  MoveL 6051 to (232.86, 162.69, 88.06) mm, rotated rx 180 ry 0 rz 180 deg; joints [-65.874, 60.657, -79.327, 67.008, 97.518, 17.138]
  Call Extruder(269.01860)
  MoveL 6052 to (232.62, 162.8, 88.06) mm, rotated rx 180 ry 0 rz 180 deg; joints [-65.961, 60.657, -79.327, 67.092, 97.493, 17.15]
  MoveL 6053 to (232.62, 162.8, 88.06) mm, rotated rx 180 ry 0 rz 180 deg; joints [-65.961, 60.657, -79.327, 67.092, 97.493, 17.15]
  Call Extruder(269.17597)
  MoveL 6054 to (232.37, 162.91, 88.06) mm, rotated rx -180 ry 0 rz 180 deg; joints [-66.048, 60.657, -79.327, 67.176, 97.467, 17.161]
  MoveL 6055 to (232.37, 162.91, 88.06) mm, rotated rx -180 ry 0 rz 180 deg; joints [-66.048, 60.657, -79.327, 67.176, 97.467, 17.161]
  Call Extruder(269.35871)
  MoveL 6056 to (232.07, 163.02, 88.06) mm, rotated rx -180 ry 0 rz -180 deg; joints [-66.149, 60.656, -79.328, 67.274, 97.438, 17.175]
  MoveL 6057 to (232.07, 163.02, 88.06) mm, rotated rx -180 ry 0 rz -180 deg; joints [-66.149, 60.656, -79.328, 67.274, 97.438, 17.175]
  Call Extruder(269.54070)
  MoveL 6058 to (231.78, 163.15, 88.06) mm, rotated rx 180 ry 0 rz 180 deg; joints [-66.251, 60.655, -79.328, 67.372, 97.408, 17.188]
  MoveL 6059 to (231.78, 163.15, 88.06) mm, rotated rx 180 ry 0 rz 180 deg; joints [-66.251, 60.655, -79.328, 67.372, 97.408, 17.188]
  Call Extruder(269.68804)
  MoveL 6060 to (231.54, 163.24, 88.06) mm, rotated rx -180 ry 0 rz -180 deg; joints [-66.333, 60.654, -79.328, 67.452, 97.384, 17.2]
  MoveL 6061 to (231.54, 163.24, 88.06) mm, rotated rx -180 ry 0 rz -180 deg; joints [-66.333, 60.654, -79.328, 67.452, 97.384, 17.2]
  Call Extruder(269.80126)
  MoveL 6062 to (231.35, 163.3, 88.06) mm, rotated rx 180 ry 0 rz -180 deg; joints [-66.397, 60.653, -79.329, 67.513, 97.367, 17.21]
  MoveL 6063 to (231.35, 163.3, 88.06) mm, rotated rx 180 ry 0 rz -180 deg; joints [-66.397, 60.653, -79.329, 67.513, 97.367, 17.21]
  Call Extruder(269.91404)
  MoveL 6064 to (231.17, 163.36, 88.06) mm, rotated rx 180 ry 0 rz -180 deg; joints [-66.46, 60.651, -79.33, 67.574, 97.349, 17.22]
  MoveL 6065 to (231.17, 163.36, 88.06) mm, rotated rx 180 ry 0 rz -180 deg; joints [-66.46, 60.651, -79.33, 67.574, 97.349, 17.22]
  Call Extruder(270.02637)
  MoveL 6066 to (230.98, 163.42, 88.06) mm, rotated rx -180 ry 0 rz 180 deg; joints [-66.524, 60.65, -79.331, 67.636, 97.331, 17.23]
  MoveL 6067 to (230.98, 163.42, 88.06) mm, rotated rx -180 ry 0 rz 180 deg; joints [-66.524, 60.65, -79.331, 67.636, 97.331, 17.23]
  Call Extruder(270.13826)
  MoveL 6068 to (230.79, 163.48, 88.06) mm, rotated rx -180 ry 0 rz 180 deg; joints [-66.587, 60.648, -79.331, 67.697, 97.313, 17.24]
  MoveL 6069 to (230.79, 163.48, 88.06) mm, rotated rx -180 ry 0 rz 180 deg; joints [-66.587, 60.648, -79.331, 67.697, 97.313, 17.24]
  Call Extruder(270.25966)
  MoveL 6070 to (230.58, 163.55, 88.06) mm, rotated rx -180 ry 0 rz -180 deg; joints [-66.656, 60.646, -79.332, 67.764, 97.293, 17.251]
  MoveL 6071 to (230.58, 163.55, 88.06) mm, rotated rx -180 ry 0 rz -180 deg; joints [-66.656, 60.646, -79.332, 67.764, 97.293, 17.251]
  Call Extruder(270.39048)
  MoveL 6072 to (230.36, 163.62, 88.06) mm, rotated rx -180 ry 0 rz 180 deg; joints [-66.731, 60.644, -79.333, 67.836, 97.272, 17.263]
  MoveL 6073 to (230.36, 163.62, 88.06) mm, rotated rx -180 ry 0 rz 180 deg; joints [-66.731, 60.644, -79.333, 67.836, 97.272, 17.263]
  Call Extruder(270.52072)
  MoveL 6074 to (230.14, 163.68, 88.06) mm, rotated rx 180 ry 0 rz 180 deg; joints [-66.805, 60.642, -79.334, 67.908, 97.251, 17.275]
  MoveL 6075 to (230.14, 163.68, 88.06) mm, rotated rx 180 ry 0 rz 180 deg; joints [-66.805, 60.642, -79.334, 67.908, 97.251, 17.275]
  Call Extruder(270.65041)
  MoveL 6076 to (229.91, 163.75, 88.06) mm, rotated rx 180 ry 0 rz -180 deg; joints [-66.88, 60.64, -79.335, 67.981, 97.23, 17.287]
  MoveL 6077 to (229.91, 163.75, 88.06) mm, rotated rx 180 ry 0 rz -180 deg; joints [-66.88, 60.64, -79.335, 67.981, 97.23, 17.287]
  Call Extruder(270.77952)
  MoveL 6078 to (229.69, 163.82, 88.06) mm, rotated rx -180 ry 0 rz 180 deg; joints [-66.955, 60.638, -79.336, 68.053, 97.209, 17.299]
  MoveL 6079 to (229.69, 163.82, 88.06) mm, rotated rx -180 ry 0 rz 180 deg; joints [-66.955, 60.638, -79.336, 68.053, 97.209, 17.299]
  Call Extruder(270.89460)
  MoveL 6080 to (229.48, 163.86, 88.06) mm, rotated rx 180 ry 0 rz 180 deg; joints [-67.021, 60.635, -79.338, 68.117, 97.191, 17.311]
  MoveL 6081 to (229.48, 163.86, 88.06) mm, rotated rx 180 ry 0 rz 180 deg; joints [-67.021, 60.635, -79.338, 68.117, 97.191, 17.311]
  Call Extruder(271.00922)
  MoveL 6082 to (229.28, 163.91, 88.06) mm, rotated rx -180 ry 0 rz 180 deg; joints [-67.087, 60.632, -79.339, 68.181, 97.173, 17.323]
  MoveL 6083 to (229.28, 163.91, 88.06) mm, rotated rx -180 ry 0 rz 180 deg; joints [-67.087, 60.632, -79.339, 68.181, 97.173, 17.323]
  Call Extruder(271.12339)
  MoveL 6084 to (229.08, 163.95, 88.06) mm, rotated rx 180 ry 0 rz -180 deg; joints [-67.153, 60.628, -79.341, 68.246, 97.155, 17.336]
  MoveL 6085 to (229.08, 163.95, 88.06) mm, rotated rx 180 ry 0 rz -180 deg; joints [-67.153, 60.628, -79.341, 68.246, 97.155, 17.336]
  Call Extruder(271.23711)
  MoveL 6086 to (228.87, 164, 88.06) mm, rotated rx 180 ry 0 rz -180 deg; joints [-67.22, 60.625, -79.342, 68.31, 97.137, 17.348]
  MoveL 6087 to (228.87, 164, 88.06) mm, rotated rx 180 ry 0 rz -180 deg; joints [-67.22, 60.625, -79.342, 68.31, 97.137, 17.348]
  Call Extruder(271.36253)
  MoveL 6088 to (228.64, 164.04, 88.06) mm, rotated rx -180 ry 0 rz -180 deg; joints [-67.293, 60.622, -79.344, 68.381, 97.118, 17.362]
  MoveL 6089 to (228.64, 164.04, 88.06) mm, rotated rx -180 ry 0 rz -180 deg; joints [-67.293, 60.622, -79.344, 68.381, 97.118, 17.362]
  Call Extruder(271.49950)
  MoveL 6090 to (228.4, 164.09, 88.06) mm, rotated rx -180 ry 0 rz -180 deg; joints [-67.373, 60.618, -79.346, 68.459, 97.096, 17.377]
  MoveL 6091 to (228.4, 164.09, 88.06) mm, rotated rx -180 ry 0 rz -180 deg; joints [-67.373, 60.618, -79.346, 68.459, 97.096, 17.377]
  Call Extruder(271.63587)
  MoveL 6092 to (228.15, 164.14, 88.06) mm, rotated rx -180 ry 0 rz 180 deg; joints [-67.453, 60.614, -79.348, 68.537, 97.074, 17.392]
  MoveL 6093 to (228.15, 164.14, 88.06) mm, rotated rx -180 ry 0 rz 180 deg; joints [-67.453, 60.614, -79.348, 68.537, 97.074, 17.392]
  Call Extruder(271.77163)
  MoveL 6094 to (227.9, 164.19, 88.06) mm, rotated rx -180 ry 0 rz -180 deg; joints [-67.534, 60.61, -79.35, 68.615, 97.052, 17.407]
  MoveL 6095 to (227.9, 164.19, 88.06) mm, rotated rx -180 ry 0 rz -180 deg; joints [-67.534, 60.61, -79.35, 68.615, 97.052, 17.407]
  Call Extruder(271.90678)
  MoveL 6096 to (227.65, 164.24, 88.06) mm, rotated rx -180 ry 0 rz 180 deg; joints [-67.614, 60.605, -79.352, 68.693, 97.03, 17.422]
  MoveL 6097 to (227.65, 164.24, 88.06) mm, rotated rx -180 ry 0 rz 180 deg; joints [-67.614, 60.605, -79.352, 68.693, 97.03, 17.422]
  Call Extruder(272.04131)
  MoveL 6098 to (227.4, 164.29, 88.06) mm, rotated rx -180 ry 0 rz 180 deg; joints [-67.695, 60.602, -79.354, 68.771, 97.008, 17.437]
  MoveL 6099 to (227.4, 164.29, 88.06) mm, rotated rx -180 ry 0 rz 180 deg; joints [-67.695, 60.602, -79.354, 68.771, 97.008, 17.437]
  Call Extruder(272.17524)
  MoveL 6100 to (227.15, 164.34, 88.06) mm, rotated rx 180 ry 0 rz -180 deg; joints [-67.775, 60.598, -79.355, 68.848, 96.986, 17.452]
  MoveL 6101 to (227.15, 164.34, 88.06) mm, rotated rx 180 ry 0 rz -180 deg; joints [-67.775, 60.598, -79.355, 68.848, 96.986, 17.452]
  Call Extruder(272.32310)
  MoveL 6102 to (226.87, 164.39, 88.06) mm, rotated rx 180 ry 0 rz 180 deg; joints [-67.864, 60.593, -79.358, 68.935, 96.962, 17.469]
  MoveL 6103 to (226.87, 164.39, 88.06) mm, rotated rx 180 ry 0 rz 180 deg; joints [-67.864, 60.593, -79.358, 68.935, 96.962, 17.469]
  Call Extruder(272.48484)
  MoveL 6104 to (226.57, 164.44, 88.06) mm, rotated rx -180 ry 0 rz -180 deg; joints [-67.961, 60.587, -79.36, 69.029, 96.936, 17.488]
  MoveL 6105 to (226.57, 164.44, 88.06) mm, rotated rx -180 ry 0 rz -180 deg; joints [-67.961, 60.587, -79.36, 69.029, 96.936, 17.488]
  Call Extruder(272.64586)
  MoveL 6106 to (226.26, 164.49, 88.06) mm, rotated rx -180 ry 0 rz -180 deg; joints [-68.059, 60.581, -79.363, 69.124, 96.91, 17.507]
  MoveL 6107 to (226.26, 164.49, 88.06) mm, rotated rx -180 ry 0 rz -180 deg; joints [-68.059, 60.581, -79.363, 69.124, 96.91, 17.507]
  Call Extruder(272.80614)
  MoveL 6108 to (225.96, 164.53, 88.06) mm, rotated rx -180 ry 0 rz 180 deg; joints [-68.156, 60.576, -79.366, 69.219, 96.883, 17.526]
  MoveL 6109 to (225.96, 164.53, 88.06) mm, rotated rx -180 ry 0 rz 180 deg; joints [-68.156, 60.576, -79.366, 69.219, 96.883, 17.526]
  Call Extruder(272.96570)
  MoveL 6110 to (225.65, 164.58, 88.06) mm, rotated rx -180 ry 0 rz 180 deg; joints [-68.254, 60.57, -79.368, 69.313, 96.857, 17.545]
  MoveL 6111 to (225.65, 164.58, 88.06) mm, rotated rx -180 ry 0 rz 180 deg; joints [-68.254, 60.57, -79.368, 69.313, 96.857, 17.545]
  Call Extruder(273.12452)
  MoveL 6112 to (225.34, 164.63, 88.06) mm, rotated rx 180 ry 0 rz 180 deg; joints [-68.351, 60.565, -79.371, 69.408, 96.83, 17.564]
  MoveL 6113 to (225.34, 164.63, 88.06) mm, rotated rx 180 ry 0 rz 180 deg; joints [-68.351, 60.565, -79.371, 69.408, 96.83, 17.564]
  Call Extruder(273.30319)
  MoveL 6114 to (225, 164.68, 88.06) mm, rotated rx 180 ry 0 rz 180 deg; joints [-68.461, 60.558, -79.374, 69.515, 96.801, 17.586]
  MoveL 6115 to (225, 164.68, 88.06) mm, rotated rx 180 ry 0 rz 180 deg; joints [-68.461, 60.558, -79.374, 69.515, 96.801, 17.586]
  Call Extruder(273.50164)
  MoveL 6116 to (224.61, 164.72, 88.06) mm, rotated rx -180 ry 0 rz 180 deg; joints [-68.583, 60.55, -79.378, 69.633, 96.768, 17.611]
  MoveL 6117 to (224.61, 164.72, 88.06) mm, rotated rx -180 ry 0 rz 180 deg; joints [-68.583, 60.55, -79.378, 69.633, 96.768, 17.611]
  Call Extruder(273.69921)
  MoveL 6118 to (224.22, 164.77, 88.06) mm, rotated rx -180 ry 0 rz 180 deg; joints [-68.706, 60.542, -79.382, 69.752, 96.735, 17.636]
  MoveL 6119 to (224.22, 164.77, 88.06) mm, rotated rx -180 ry 0 rz 180 deg; joints [-68.706, 60.542, -79.382, 69.752, 96.735, 17.636]
  Call Extruder(273.89592)
  MoveL 6120 to (223.84, 164.82, 88.06) mm, rotated rx 180 ry 0 rz 180 deg; joints [-68.828, 60.534, -79.386, 69.871, 96.702, 17.661]
  MoveL 6121 to (223.84, 164.82, 88.06) mm, rotated rx 180 ry 0 rz 180 deg; joints [-68.828, 60.534, -79.386, 69.871, 96.702, 17.661]
  Call Extruder(274.09176)
  MoveL 6122 to (223.45, 164.86, 88.06) mm, rotated rx -180 ry 0 rz 180 deg; joints [-68.951, 60.526, -79.389, 69.989, 96.669, 17.686]
  MoveL 6123 to (223.45, 164.86, 88.06) mm, rotated rx -180 ry 0 rz 180 deg; joints [-68.951, 60.526, -79.389, 69.989, 96.669, 17.686]
  Call Extruder(274.38712)
  MoveL 6124 to (222.86, 164.91, 88.06) mm, rotated rx -180 ry 0 rz 180 deg; joints [-69.135, 60.512, -79.396, 70.168, 96.62, 17.725]
  MoveL 6125 to (222.86, 164.91, 88.06) mm, rotated rx -180 ry 0 rz 180 deg; joints [-69.135, 60.512, -79.396, 70.168, 96.62, 17.725]
  Call Extruder(274.68114)
  MoveL 6126 to (222.27, 164.95, 88.06) mm, rotated rx 180 ry 0 rz 180 deg; joints [-69.319, 60.498, -79.402, 70.347, 96.57, 17.765]
  MoveL 6127 to (222.27, 164.95, 88.06) mm, rotated rx 180 ry 0 rz 180 deg; joints [-69.319, 60.498, -79.402, 70.347, 96.57, 17.765]
  Call Extruder(274.97384)
  MoveL 6128 to (221.68, 165, 88.06) mm, rotated rx -180 ry 0 rz 180 deg; joints [-69.504, 60.485, -79.408, 70.526, 96.52, 17.803]
  MoveL 6129 to (221.68, 165, 88.06) mm, rotated rx -180 ry 0 rz 180 deg; joints [-69.504, 60.485, -79.408, 70.526, 96.52, 17.803]
  Call Extruder(275.54729)
  MoveL 6130 to (220.52, 165.05, 88.06) mm, rotated rx -180 ry 0 rz 180 deg; joints [-69.864, 60.455, -79.422, 70.876, 96.424, 17.884]
  MoveL 6131 to (220.52, 165.05, 88.06) mm, rotated rx -180 ry 0 rz 180 deg; joints [-69.864, 60.455, -79.422, 70.876, 96.424, 17.884]
  Call Extruder(276.26129)
  MoveL 6132 to (219.06, 165.09, 88.06) mm, rotated rx -180 ry 0 rz 180 deg; joints [-70.315, 60.418, -79.44, 71.313, 96.303, 17.984]
  Call Extruder(393.10803)
  MoveL 6133 to (-19.06, 165.09, 88.06) mm, rotated rx -180 ry 0 rz 180 deg; joints [-137.325, 65.34, -75.969, 136.831, 82.206, 7.25]
  Call Extruder(393.53664)
  MoveL 6134 to (-19.94, 165.07, 88.06) mm, rotated rx -180 ry 0 rz 180 deg; joints [-137.467, 65.379, -75.929, 136.98, 82.246, 7.176]
  MoveL 6135 to (-19.94, 165.07, 88.06) mm, rotated rx -180 ry 0 rz 180 deg; joints [-137.467, 65.379, -75.929, 136.98, 82.246, 7.176]
  Call Extruder(394.11009)
  MoveL 6136 to (-21.1, 165.03, 88.06) mm, rotated rx 180 ry 0 rz 180 deg; joints [-137.659, 65.429, -75.876, 137.182, 82.298, 7.079]
  MoveL 6137 to (-21.1, 165.03, 88.06) mm, rotated rx 180 ry 0 rz 180 deg; joints [-137.659, 65.429, -75.876, 137.182, 82.298, 7.079]
  Call Extruder(394.54439)
  MoveL 6138 to (-21.97, 164.98, 88.06) mm, rotated rx 180 ry 0 rz 180 deg; joints [-137.804, 65.467, -75.836, 137.335, 82.337, 7.006]
  MoveL 6139 to (-21.97, 164.98, 88.06) mm, rotated rx 180 ry 0 rz 180 deg; joints [-137.804, 65.467, -75.836, 137.335, 82.337, 7.006]
  Call Extruder(394.83842)
  MoveL 6140 to (-22.56, 164.93, 88.06) mm, rotated rx -180 ry 0 rz 180 deg; joints [-137.905, 65.492, -75.81, 137.44, 82.363, 6.958]
  MoveL 6141 to (-22.56, 164.93, 88.06) mm, rotated rx -180 ry 0 rz 180 deg; joints [-137.905, 65.492, -75.81, 137.44, 82.363, 6.958]
  Call Extruder(395.13378)
  MoveL 6142 to (-23.15, 164.89, 88.06) mm, rotated rx -180 ry 0 rz -180 deg; joints [-138.004, 65.517, -75.783, 137.544, 82.388, 6.91]
  MoveL 6143 to (-23.15, 164.89, 88.06) mm, rotated rx -180 ry 0 rz -180 deg; joints [-138.004, 65.517, -75.783, 137.544, 82.388, 6.91]
  Call Extruder(395.37999)
  MoveL 6144 to (-23.64, 164.84, 88.06) mm, rotated rx -180 ry 0 rz -180 deg; joints [-138.088, 65.537, -75.762, 137.632, 82.409, 6.87]
  MoveL 6145 to (-23.64, 164.84, 88.06) mm, rotated rx -180 ry 0 rz -180 deg; joints [-138.088, 65.537, -75.762, 137.632, 82.409, 6.87]
  Call Extruder(395.57670)
  MoveL 6146 to (-24.03, 164.79, 88.06) mm, rotated rx -180 ry 0 rz 180 deg; joints [-138.156, 65.553, -75.745, 137.703, 82.425, 6.839]
  MoveL 6147 to (-24.03, 164.79, 88.06) mm, rotated rx -180 ry 0 rz 180 deg; joints [-138.156, 65.553, -75.745, 137.703, 82.425, 6.839]
  Call Extruder(395.77427)
  MoveL 6148 to (-24.42, 164.75, 88.06) mm, rotated rx 180 ry 0 rz 180 deg; joints [-138.224, 65.568, -75.728, 137.774, 82.441, 6.808]
  MoveL 6149 to (-24.42, 164.75, 88.06) mm, rotated rx 180 ry 0 rz 180 deg; joints [-138.224, 65.568, -75.728, 137.774, 82.441, 6.808]
  Call Extruder(395.97271)
  MoveL 6150 to (-24.8, 164.7, 88.06) mm, rotated rx -180 ry 0 rz 180 deg; joints [-138.292, 65.584, -75.711, 137.844, 82.457, 6.777]
  MoveL 6151 to (-24.8, 164.7, 88.06) mm, rotated rx -180 ry 0 rz 180 deg; joints [-138.292, 65.584, -75.711, 137.844, 82.457, 6.777]
  Call Extruder(396.17202)
  MoveL 6152 to (-25.19, 164.66, 88.06) mm, rotated rx -180 ry 0 rz 180 deg; joints [-138.359, 65.6, -75.694, 137.915, 82.473, 6.746]
  MoveL 6153 to (-25.19, 164.66, 88.06) mm, rotated rx -180 ry 0 rz 180 deg; joints [-138.359, 65.6, -75.694, 137.915, 82.473, 6.746]
  Call Extruder(396.33085)
  MoveL 6154 to (-25.5, 164.61, 88.06) mm, rotated rx -180 ry 0 rz -180 deg; joints [-138.415, 65.611, -75.681, 137.973, 82.485, 6.722]
  MoveL 6155 to (-25.5, 164.61, 88.06) mm, rotated rx -180 ry 0 rz -180 deg; joints [-138.415, 65.611, -75.681, 137.973, 82.485, 6.722]
  Call Extruder(396.49041)
  MoveL 6156 to (-25.8, 164.56, 88.06) mm, rotated rx -180 ry 0 rz -180 deg; joints [-138.47, 65.623, -75.669, 138.03, 82.497, 6.699]
  MoveL 6157 to (-25.8, 164.56, 88.06) mm, rotated rx -180 ry 0 rz -180 deg; joints [-138.47, 65.623, -75.669, 138.03, 82.497, 6.699]
  Call Extruder(396.65070)
  MoveL 6158 to (-26.11, 164.51, 88.06) mm, rotated rx -180 ry 0 rz 180 deg; joints [-138.525, 65.635, -75.656, 138.087, 82.509, 6.675]
  MoveL 6159 to (-26.11, 164.51, 88.06) mm, rotated rx -180 ry 0 rz 180 deg; joints [-138.525, 65.635, -75.656, 138.087, 82.509, 6.675]
  Call Extruder(396.81172)
  MoveL 6160 to (-26.41, 164.46, 88.06) mm, rotated rx -180 ry 0 rz 180 deg; joints [-138.58, 65.647, -75.643, 138.145, 82.521, 6.651]
  MoveL 6161 to (-26.41, 164.46, 88.06) mm, rotated rx -180 ry 0 rz 180 deg; joints [-138.58, 65.647, -75.643, 138.145, 82.521, 6.651]
  Call Extruder(396.97346)
  MoveL 6162 to (-26.72, 164.41, 88.06) mm, rotated rx -180 ry 0 rz 180 deg; joints [-138.635, 65.659, -75.63, 138.202, 82.533, 6.627]
  MoveL 6163 to (-26.72, 164.41, 88.06) mm, rotated rx -180 ry 0 rz 180 deg; joints [-138.635, 65.659, -75.63, 138.202, 82.533, 6.627]
  Call Extruder(397.13593)
  MoveL 6164 to (-27.03, 164.37, 88.06) mm, rotated rx 180 ry 0 rz 180 deg; joints [-138.69, 65.671, -75.617, 138.259, 82.546, 6.603]
  MoveL 6165 to (-27.03, 164.37, 88.06) mm, rotated rx 180 ry 0 rz 180 deg; joints [-138.69, 65.671, -75.617, 138.259, 82.546, 6.603]
  Call Extruder(397.26986)
  MoveL 6166 to (-27.27, 164.32, 88.06) mm, rotated rx -180 ry 0 rz 180 deg; joints [-138.736, 65.68, -75.607, 138.307, 82.555, 6.584]
  MoveL 6167 to (-27.27, 164.32, 88.06) mm, rotated rx -180 ry 0 rz 180 deg; joints [-138.736, 65.68, -75.607, 138.307, 82.555, 6.584]
  Call Extruder(397.40439)
  MoveL 6168 to (-27.52, 164.27, 88.06) mm, rotated rx 180 ry 0 rz 180 deg; joints [-138.783, 65.689, -75.596, 138.355, 82.564, 6.565]
  MoveL 6169 to (-27.52, 164.27, 88.06) mm, rotated rx 180 ry 0 rz 180 deg; joints [-138.783, 65.689, -75.596, 138.355, 82.564, 6.565]
  Call Extruder(397.53954)
  MoveL 6170 to (-27.77, 164.22, 88.06) mm, rotated rx 180 ry 0 rz 180 deg; joints [-138.829, 65.699, -75.586, 138.404, 82.573, 6.546]
  MoveL 6171 to (-27.77, 164.22, 88.06) mm, rotated rx 180 ry 0 rz 180 deg; joints [-138.829, 65.699, -75.586, 138.404, 82.573, 6.546]
  Call Extruder(397.67530)
  MoveL 6172 to (-28.02, 164.17, 88.06) mm, rotated rx 180 ry 0 rz 180 deg; joints [-138.875, 65.708, -75.576, 138.451, 82.583, 6.527]
  MoveL 6173 to (-28.02, 164.17, 88.06) mm, rotated rx 180 ry 0 rz 180 deg; joints [-138.875, 65.708, -75.576, 138.451, 82.583, 6.527]
  Call Extruder(397.81166)
  MoveL 6174 to (-28.27, 164.12, 88.06) mm, rotated rx -180 ry 0 rz 180 deg; joints [-138.921, 65.717, -75.566, 138.499, 82.592, 6.508]
  MoveL 6175 to (-28.27, 164.12, 88.06) mm, rotated rx -180 ry 0 rz 180 deg; joints [-138.921, 65.717, -75.566, 138.499, 82.592, 6.508]
  Call Extruder(397.89653)
  MoveL 6176 to (-28.42, 164.09, 88.06) mm, rotated rx -180 ry 0 rz 180 deg; joints [-138.95, 65.723, -75.559, 138.529, 82.598, 6.496]
  Set speed (130.0 mm/s)
  MoveL 6177 to (-31.76, 163.31, 88.06) mm, rotated rx -180 ry 0 rz -180 deg; joints [-139.581, 65.843, -75.425, 139.183, 82.719, 6.247]
  MoveL 6178 to (-31.76, 163.31, 97.46) mm, rotated rx -180 ry 0 rz 180 deg; joints [-139.581, 67.208, -77.308, 139.139, 82.328, 6.588]
  Call Extruder(395.89653)
  Set speed (40.0 mm/s)
  MoveL 6179 to (-31.76, 163.31, 97.46) mm, rotated rx -180 ry 0 rz 180 deg; joints [-139.581, 67.208, -77.308, 139.139, 82.328, 6.588]
  Call Extruder(0.00000)
  Set speed (130.0 mm/s)
  MoveL 6180 to (-31.64, 163.21, 97.46) mm, rotated rx 180 ry 0 rz 180 deg; joints [-139.581, 67.199, -77.319, 139.137, 82.313, 6.601]
  Call Extruder(2.00000)
  Set speed (40.0 mm/s)
  MoveL 6181 to (-31.64, 163.21, 97.46) mm, rotated rx 180 ry 0 rz 180 deg; joints [-139.581, 67.199, -77.319, 139.137, 82.313, 6.601]
  Set speed (30.0 mm/s)
  MoveL 6182 to (-31.64, 163.21, 97.46) mm, rotated rx 180 ry 0 rz 180 deg; joints [-139.581, 67.199, -77.319, 139.137, 82.313, 6.601]
  Call Extruder(2.18198)
  MoveL 6183 to (-31.93, 163.09, 97.46) mm, rotated rx 180 ry 0 rz 180 deg; joints [-139.645, 67.208, -77.309, 139.203, 82.319, 6.58]
  MoveL 6184 to (-31.93, 163.09, 97.46) mm, rotated rx 180 ry 0 rz 180 deg; joints [-139.645, 67.208, -77.309, 139.203, 82.319, 6.58]
  Call Extruder(2.36471)
  MoveL 6185 to (-32.22, 162.96, 97.46) mm, rotated rx -180 ry 0 rz -180 deg; joints [-139.709, 67.216, -77.299, 139.268, 82.326, 6.56]
  MoveL 6186 to (-32.22, 162.96, 97.46) mm, rotated rx -180 ry 0 rz -180 deg; joints [-139.709, 67.216, -77.299, 139.268, 82.326, 6.56]
  Call Extruder(2.53513)
  MoveL 6187 to (-32.49, 162.85, 97.46) mm, rotated rx -180 ry 0 rz 180 deg; joints [-139.768, 67.224, -77.29, 139.329, 82.332, 6.541]
  MoveL 6188 to (-32.49, 162.85, 97.46) mm, rotated rx -180 ry 0 rz 180 deg; joints [-139.768, 67.224, -77.29, 139.329, 82.332, 6.541]
  Call Extruder(2.69310)
  MoveL 6189 to (-32.74, 162.74, 97.46) mm, rotated rx 180 ry 0 rz 180 deg; joints [-139.823, 67.232, -77.282, 139.386, 82.337, 6.523]
  MoveL 6190 to (-32.74, 162.74, 97.46) mm, rotated rx 180 ry 0 rz 180 deg; joints [-139.823, 67.232, -77.282, 139.386, 82.337, 6.523]
  Call Extruder(2.85168)
  MoveL 6191 to (-32.99, 162.64, 97.46) mm, rotated rx -180 ry 0 rz -180 deg; joints [-139.878, 67.239, -77.274, 139.443, 82.343, 6.506]
  MoveL 6192 to (-32.99, 162.64, 97.46) mm, rotated rx -180 ry 0 rz -180 deg; joints [-139.878, 67.239, -77.274, 139.443, 82.343, 6.506]
  Call Extruder(3.05785)
  MoveL 6193 to (-33.29, 162.46, 97.46) mm, rotated rx -180 ry 0 rz -180 deg; joints [-139.953, 67.246, -77.266, 139.519, 82.346, 6.486]
  MoveL 6194 to (-33.29, 162.46, 97.46) mm, rotated rx -180 ry 0 rz -180 deg; joints [-139.953, 67.246, -77.266, 139.519, 82.346, 6.486]
  Call Extruder(3.26479)
  MoveL 6195 to (-33.6, 162.29, 97.46) mm, rotated rx -180 ry 0 rz -180 deg; joints [-140.028, 67.253, -77.258, 139.595, 82.349, 6.466]
  MoveL 6196 to (-33.6, 162.29, 97.46) mm, rotated rx -180 ry 0 rz -180 deg; joints [-140.028, 67.253, -77.258, 139.595, 82.349, 6.466]
  Call Extruder(3.47251)
  MoveL 6197 to (-33.9, 162.11, 97.46) mm, rotated rx 180 ry 0 rz 180 deg; joints [-140.103, 67.261, -77.25, 139.672, 82.352, 6.446]
  MoveL 6198 to (-33.9, 162.11, 97.46) mm, rotated rx 180 ry 0 rz 180 deg; joints [-140.103, 67.261, -77.25, 139.672, 82.352, 6.446]
  Call Extruder(3.68101)
  MoveL 6199 to (-34.21, 161.94, 97.46) mm, rotated rx 180 ry 0 rz 180 deg; joints [-140.178, 67.268, -77.242, 139.748, 82.356, 6.426]
  MoveL 6200 to (-34.21, 161.94, 97.46) mm, rotated rx 180 ry 0 rz 180 deg; joints [-140.178, 67.268, -77.242, 139.748, 82.356, 6.426]
  Call Extruder(3.86055)
  MoveL 6201 to (-34.45, 161.76, 97.46) mm, rotated rx 180 ry 0 rz 180 deg; joints [-140.244, 67.272, -77.237, 139.815, 82.356, 6.411]
  MoveL 6202 to (-34.45, 161.76, 97.46) mm, rotated rx 180 ry 0 rz 180 deg; joints [-140.244, 67.272, -77.237, 139.815, 82.356, 6.411]
  Call Extruder(4.19399)
  MoveL 6203 to (-34.9, 161.43, 97.46) mm, rotated rx 180 ry 0 rz 180 deg; joints [-140.366, 67.281, -77.227, 139.939, 82.355, 6.383]
  MoveL 6204 to (-34.9, 161.43, 97.46) mm, rotated rx 180 ry 0 rz 180 deg; joints [-140.366, 67.281, -77.227, 139.939, 82.355, 6.383]
  Call Extruder(4.52861)
  MoveL 6205 to (-35.35, 161.1, 97.46) mm, rotated rx -180 ry 0 rz -180 deg; joints [-140.489, 67.289, -77.218, 140.064, 82.355, 6.355]
  Call Extruder(5.35652)
  MoveL 6206 to (-36.39, 160.19, 97.46) mm, rotated rx -180 ry 0 rz 180 deg; joints [-140.797, 67.302, -77.203, 140.375, 82.343, 6.295]
  Call Extruder(6.18445)
  MoveL 6207 to (-37.3, 159.15, 97.46) mm, rotated rx -180 ry 0 rz 180 deg; joints [-141.109, 67.306, -77.199, 140.689, 82.315, 6.249]
  Call Extruder(6.35176)
  MoveL 6208 to (-37.47, 158.93, 97.46) mm, rotated rx -180 ry 0 rz -180 deg; joints [-141.172, 67.305, -77.2, 140.752, 82.306, 6.242]
  MoveL 6209 to (-37.47, 158.93, 97.46) mm, rotated rx -180 ry 0 rz -180 deg; joints [-141.172, 67.305, -77.2, 140.752, 82.306, 6.242]
  Call Extruder(6.68519)
  MoveL 6210 to (-37.8, 158.48, 97.46) mm, rotated rx 180 ry 0 rz 180 deg; joints [-141.298, 67.303, -77.202, 140.878, 82.29, 6.227]
  MoveL 6211 to (-37.8, 158.48, 97.46) mm, rotated rx 180 ry 0 rz 180 deg; joints [-141.298, 67.303, -77.202, 140.878, 82.29, 6.227]
  Call Extruder(7.01743)
  MoveL 6212 to (-38.12, 158.03, 97.46) mm, rotated rx 180 ry 0 rz 180 deg; joints [-141.424, 67.302, -77.204, 141.004, 82.274, 6.212]
  MoveL 6213 to (-38.12, 158.03, 97.46) mm, rotated rx 180 ry 0 rz 180 deg; joints [-141.424, 67.302, -77.204, 141.004, 82.274, 6.212]
  Call Extruder(7.13511)
  MoveL 6214 to (-38.22, 157.85, 97.46) mm, rotated rx 180 ry 0 rz 180 deg; joints [-141.468, 67.3, -77.206, 141.048, 82.266, 6.209]
  MoveL 6215 to (-38.22, 157.85, 97.46) mm, rotated rx 180 ry 0 rz 180 deg; joints [-141.468, 67.3, -77.206, 141.048, 82.266, 6.209]
  Call Extruder(7.34283)
  MoveL 6216 to (-38.4, 157.55, 97.46) mm, rotated rx -180 ry 0 rz 180 deg; joints [-141.547, 67.297, -77.209, 141.126, 82.253, 6.202]
  MoveL 6217 to (-38.4, 157.55, 97.46) mm, rotated rx -180 ry 0 rz 180 deg; joints [-141.547, 67.297, -77.209, 141.126, 82.253, 6.202]
  Call Extruder(7.54978)
  MoveL 6218 to (-38.57, 157.25, 97.46) mm, rotated rx -180 ry 0 rz 180 deg; joints [-141.625, 67.294, -77.213, 141.204, 82.239, 6.196]
  MoveL 6219 to (-38.57, 157.25, 97.46) mm, rotated rx -180 ry 0 rz 180 deg; joints [-141.625, 67.294, -77.213, 141.204, 82.239, 6.196]
  Call Extruder(7.75595)
  MoveL 6220 to (-38.75, 156.94, 97.46) mm, rotated rx 180 ry 0 rz 180 deg; joints [-141.704, 67.291, -77.216, 141.283, 82.226, 6.189]
  MoveL 6221 to (-38.75, 156.94, 97.46) mm, rotated rx 180 ry 0 rz 180 deg; joints [-141.704, 67.291, -77.216, 141.283, 82.226, 6.189]
  Call Extruder(7.93762)
  MoveL 6222 to (-38.89, 156.67, 97.46) mm, rotated rx 180 ry 0 rz -180 deg; joints [-141.773, 67.287, -77.22, 141.351, 82.212, 6.185]
  MoveL 6223 to (-38.89, 156.67, 97.46) mm, rotated rx 180 ry 0 rz -180 deg; joints [-141.773, 67.287, -77.22, 141.351, 82.212, 6.185]
  Call Extruder(8.09561)
  MoveL 6224 to (-39, 156.42, 97.46) mm, rotated rx -180 ry 0 rz 180 deg; joints [-141.832, 67.283, -77.225, 141.41, 82.199, 6.182]
  MoveL 6225 to (-39, 156.42, 97.46) mm, rotated rx -180 ry 0 rz 180 deg; joints [-141.832, 67.283, -77.225, 141.41, 82.199, 6.182]
  Call Extruder(8.25299)
  MoveL 6226 to (-39.11, 156.17, 97.46) mm, rotated rx -180 ry 0 rz 180 deg; joints [-141.891, 67.279, -77.229, 141.469, 82.185, 6.18]
  MoveL 6227 to (-39.11, 156.17, 97.46) mm, rotated rx -180 ry 0 rz 180 deg; joints [-141.891, 67.279, -77.229, 141.469, 82.185, 6.18]
  Call Extruder(8.43571)
  MoveL 6228 to (-39.22, 155.87, 97.46) mm, rotated rx -180 ry 0 rz 180 deg; joints [-141.96, 67.274, -77.235, 141.537, 82.169, 6.177]
  MoveL 6229 to (-39.22, 155.87, 97.46) mm, rotated rx -180 ry 0 rz 180 deg; joints [-141.96, 67.274, -77.235, 141.537, 82.169, 6.177]
  Call Extruder(8.61768)
  MoveL 6230 to (-39.35, 155.58, 97.46) mm, rotated rx -180 ry 0 rz 180 deg; joints [-142.029, 67.269, -77.241, 141.605, 82.154, 6.174]
  MoveL 6231 to (-39.35, 155.58, 97.46) mm, rotated rx -180 ry 0 rz 180 deg; joints [-142.029, 67.269, -77.241, 141.605, 82.154, 6.174]
  Call Extruder(8.76501)
  MoveL 6232 to (-39.44, 155.34, 97.46) mm, rotated rx -180 ry 0 rz 180 deg; joints [-142.085, 67.264, -77.246, 141.66, 82.14, 6.173]
  MoveL 6233 to (-39.44, 155.34, 97.46) mm, rotated rx -180 ry 0 rz 180 deg; joints [-142.085, 67.264, -77.246, 141.66, 82.14, 6.173]
  Call Extruder(8.87824)
  MoveL 6234 to (-39.5, 155.15, 97.46) mm, rotated rx -180 ry 0 rz 180 deg; joints [-142.127, 67.26, -77.251, 141.702, 82.129, 6.172]
  MoveL 6235 to (-39.5, 155.15, 97.46) mm, rotated rx -180 ry 0 rz 180 deg; joints [-142.127, 67.26, -77.251, 141.702, 82.129, 6.172]
  Call Extruder(8.99103)
  MoveL 6236 to (-39.56, 154.97, 97.46) mm, rotated rx -180 ry 0 rz -180 deg; joints [-142.169, 67.256, -77.255, 141.744, 82.118, 6.172]
  MoveL 6237 to (-39.56, 154.97, 97.46) mm, rotated rx -180 ry 0 rz -180 deg; joints [-142.169, 67.256, -77.255, 141.744, 82.118, 6.172]
  Call Extruder(9.10338)
  MoveL 6238 to (-39.62, 154.78, 97.46) mm, rotated rx -180 ry 0 rz 180 deg; joints [-142.212, 67.252, -77.26, 141.785, 82.106, 6.171]
  MoveL 6239 to (-39.62, 154.78, 97.46) mm, rotated rx -180 ry 0 rz 180 deg; joints [-142.212, 67.252, -77.26, 141.785, 82.106, 6.171]
  Call Extruder(9.21528)
  MoveL 6240 to (-39.68, 154.59, 97.46) mm, rotated rx -180 ry 0 rz -180 deg; joints [-142.254, 67.248, -77.264, 141.827, 82.095, 6.171]
  MoveL 6241 to (-39.68, 154.59, 97.46) mm, rotated rx -180 ry 0 rz -180 deg; joints [-142.254, 67.248, -77.264, 141.827, 82.095, 6.171]
  Call Extruder(9.33668)
  MoveL 6242 to (-39.75, 154.38, 97.46) mm, rotated rx -180 ry 0 rz -180 deg; joints [-142.3, 67.243, -77.269, 141.872, 82.083, 6.17]
  MoveL 6243 to (-39.75, 154.38, 97.46) mm, rotated rx -180 ry 0 rz -180 deg; joints [-142.3, 67.243, -77.269, 141.872, 82.083, 6.17]
  Call Extruder(9.46747)
  MoveL 6244 to (-39.81, 154.16, 97.46) mm, rotated rx -180 ry 0 rz 180 deg; joints [-142.35, 67.238, -77.275, 141.921, 82.069, 6.17]
  MoveL 6245 to (-39.81, 154.16, 97.46) mm, rotated rx -180 ry 0 rz 180 deg; joints [-142.35, 67.238, -77.275, 141.921, 82.069, 6.17]
  Call Extruder(9.59770)
  MoveL 6246 to (-39.88, 153.94, 97.46) mm, rotated rx 180 ry 0 rz 180 deg; joints [-142.399, 67.233, -77.28, 141.97, 82.055, 6.17]
  MoveL 6247 to (-39.88, 153.94, 97.46) mm, rotated rx 180 ry 0 rz 180 deg; joints [-142.399, 67.233, -77.28, 141.97, 82.055, 6.17]
  Call Extruder(9.72737)
  MoveL 6248 to (-39.95, 153.71, 97.46) mm, rotated rx -180 ry 0 rz 180 deg; joints [-142.449, 67.228, -77.286, 142.019, 82.042, 6.17]
  MoveL 6249 to (-39.95, 153.71, 97.46) mm, rotated rx -180 ry 0 rz 180 deg; joints [-142.449, 67.228, -77.286, 142.019, 82.042, 6.17]
  Call Extruder(9.85647)
  MoveL 6250 to (-40.02, 153.49, 97.46) mm, rotated rx 180 ry 0 rz -180 deg; joints [-142.498, 67.223, -77.291, 142.068, 82.028, 6.169]
  MoveL 6251 to (-40.02, 153.49, 97.46) mm, rotated rx 180 ry 0 rz -180 deg; joints [-142.498, 67.223, -77.291, 142.068, 82.028, 6.169]
  Call Extruder(9.97155)
  MoveL 6252 to (-40.06, 153.28, 97.46) mm, rotated rx -180 ry 0 rz 180 deg; joints [-142.541, 67.218, -77.297, 142.11, 82.014, 6.17]
  MoveL 6253 to (-40.06, 153.28, 97.46) mm, rotated rx -180 ry 0 rz 180 deg; joints [-142.541, 67.218, -77.297, 142.11, 82.014, 6.17]
  Call Extruder(10.08619)
  MoveL 6254 to (-40.11, 153.08, 97.46) mm, rotated rx -180 ry 0 rz 180 deg; joints [-142.584, 67.213, -77.303, 142.152, 82.001, 6.171]
  MoveL 6255 to (-40.11, 153.08, 97.46) mm, rotated rx -180 ry 0 rz 180 deg; joints [-142.584, 67.213, -77.303, 142.152, 82.001, 6.171]
  Call Extruder(10.20037)
  MoveL 6256 to (-40.15, 152.88, 97.46) mm, rotated rx -180 ry 0 rz 180 deg; joints [-142.627, 67.207, -77.309, 142.195, 81.987, 6.172]
  MoveL 6257 to (-40.15, 152.88, 97.46) mm, rotated rx -180 ry 0 rz 180 deg; joints [-142.627, 67.207, -77.309, 142.195, 81.987, 6.172]
  Call Extruder(10.31410)
  MoveL 6258 to (-40.2, 152.67, 97.46) mm, rotated rx 180 ry 0 rz -180 deg; joints [-142.671, 67.202, -77.315, 142.237, 81.974, 6.173]
  MoveL 6259 to (-40.2, 152.67, 97.46) mm, rotated rx 180 ry 0 rz -180 deg; joints [-142.671, 67.202, -77.315, 142.237, 81.974, 6.173]
  Call Extruder(10.43952)
  MoveL 6260 to (-40.24, 152.44, 97.46) mm, rotated rx -180 ry 0 rz -180 deg; joints [-142.718, 67.196, -77.322, 142.284, 81.959, 6.174]
  MoveL 6261 to (-40.24, 152.44, 97.46) mm, rotated rx -180 ry 0 rz -180 deg; joints [-142.718, 67.196, -77.322, 142.284, 81.959, 6.174]
  Call Extruder(10.57650)
  MoveL 6262 to (-40.29, 152.2, 97.46) mm, rotated rx 180 ry 0 rz -180 deg; joints [-142.77, 67.189, -77.329, 142.335, 81.942, 6.176]
  MoveL 6263 to (-40.29, 152.2, 97.46) mm, rotated rx 180 ry 0 rz -180 deg; joints [-142.77, 67.189, -77.329, 142.335, 81.942, 6.176]
  Call Extruder(10.71287)
  MoveL 6264 to (-40.34, 151.95, 97.46) mm, rotated rx 180 ry 0 rz -180 deg; joints [-142.822, 67.182, -77.337, 142.386, 81.925, 6.177]
  MoveL 6265 to (-40.34, 151.95, 97.46) mm, rotated rx 180 ry 0 rz -180 deg; joints [-142.822, 67.182, -77.337, 142.386, 81.925, 6.177]
  Call Extruder(10.84862)
  MoveL 6266 to (-40.39, 151.7, 97.46) mm, rotated rx 180 ry 0 rz 180 deg; joints [-142.874, 67.176, -77.344, 142.437, 81.908, 6.178]
  MoveL 6267 to (-40.39, 151.7, 97.46) mm, rotated rx 180 ry 0 rz 180 deg; joints [-142.874, 67.176, -77.344, 142.437, 81.908, 6.178]
  Call Extruder(10.98377)
  MoveL 6268 to (-40.44, 151.45, 97.46) mm, rotated rx 180 ry 0 rz 180 deg; joints [-142.926, 67.169, -77.351, 142.488, 81.891, 6.18]
  MoveL 6269 to (-40.44, 151.45, 97.46) mm, rotated rx 180 ry 0 rz 180 deg; joints [-142.926, 67.169, -77.351, 142.488, 81.891, 6.18]
  Call Extruder(11.11830)
  MoveL 6270 to (-40.49, 151.2, 97.46) mm, rotated rx 180 ry 0 rz 180 deg; joints [-142.978, 67.162, -77.359, 142.539, 81.875, 6.181]
  MoveL 6271 to (-40.49, 151.2, 97.46) mm, rotated rx 180 ry 0 rz 180 deg; joints [-142.978, 67.162, -77.359, 142.539, 81.875, 6.181]
  Call Extruder(11.25223)
  MoveL 6272 to (-40.54, 150.95, 97.46) mm, rotated rx -180 ry 0 rz 180 deg; joints [-143.031, 67.156, -77.366, 142.59, 81.858, 6.182]
  MoveL 6273 to (-40.54, 150.95, 97.46) mm, rotated rx -180 ry 0 rz 180 deg; joints [-143.031, 67.156, -77.366, 142.59, 81.858, 6.182]
  Call Extruder(11.40008)
  MoveL 6274 to (-40.59, 150.67, 97.46) mm, rotated rx 180 ry 0 rz -180 deg; joints [-143.088, 67.148, -77.375, 142.646, 81.839, 6.184]
  MoveL 6275 to (-40.59, 150.67, 97.46) mm, rotated rx 180 ry 0 rz -180 deg; joints [-143.088, 67.148, -77.375, 142.646, 81.839, 6.184]
  Call Extruder(11.56181)
  MoveL 6276 to (-40.64, 150.37, 97.46) mm, rotated rx 180 ry 0 rz 180 deg; joints [-143.15, 67.139, -77.384, 142.708, 81.817, 6.186]
  MoveL 6277 to (-40.64, 150.37, 97.46) mm, rotated rx 180 ry 0 rz 180 deg; joints [-143.15, 67.139, -77.384, 142.708, 81.817, 6.186]
  Call Extruder(11.72281)
  MoveL 6278 to (-40.69, 150.06, 97.46) mm, rotated rx -180 ry 0 rz 180 deg; joints [-143.213, 67.13, -77.394, 142.769, 81.796, 6.189]
  MoveL 6279 to (-40.69, 150.06, 97.46) mm, rotated rx -180 ry 0 rz 180 deg; joints [-143.213, 67.13, -77.394, 142.769, 81.796, 6.189]
  Call Extruder(11.88308)
  MoveL 6280 to (-40.73, 149.76, 97.46) mm, rotated rx 180 ry 0 rz 180 deg; joints [-143.276, 67.122, -77.403, 142.83, 81.775, 6.191]
  MoveL 6281 to (-40.73, 149.76, 97.46) mm, rotated rx 180 ry 0 rz 180 deg; joints [-143.276, 67.122, -77.403, 142.83, 81.775, 6.191]
  Call Extruder(12.04262)
  MoveL 6282 to (-40.78, 149.45, 97.46) mm, rotated rx -180 ry 0 rz -180 deg; joints [-143.338, 67.113, -77.413, 142.891, 81.753, 6.193]
  MoveL 6283 to (-40.78, 149.45, 97.46) mm, rotated rx -180 ry 0 rz -180 deg; joints [-143.338, 67.113, -77.413, 142.891, 81.753, 6.193]
  Call Extruder(12.20144)
  MoveL 6284 to (-40.83, 149.14, 97.46) mm, rotated rx -180 ry 0 rz 180 deg; joints [-143.401, 67.104, -77.422, 142.953, 81.732, 6.195]
  MoveL 6285 to (-40.83, 149.14, 97.46) mm, rotated rx -180 ry 0 rz 180 deg; joints [-143.401, 67.104, -77.422, 142.953, 81.732, 6.195]
  Call Extruder(12.38010)
  MoveL 6286 to (-40.88, 148.8, 97.46) mm, rotated rx -180 ry 0 rz -180 deg; joints [-143.471, 67.094, -77.434, 143.022, 81.707, 6.198]
  MoveL 6287 to (-40.88, 148.8, 97.46) mm, rotated rx -180 ry 0 rz -180 deg; joints [-143.471, 67.094, -77.434, 143.022, 81.707, 6.198]
  Call Extruder(12.57854)
  MoveL 6288 to (-40.93, 148.41, 97.46) mm, rotated rx 180 ry 0 rz 180 deg; joints [-143.549, 67.082, -77.446, 143.098, 81.679, 6.202]
  MoveL 6289 to (-40.93, 148.41, 97.46) mm, rotated rx 180 ry 0 rz 180 deg; joints [-143.549, 67.082, -77.446, 143.098, 81.679, 6.202]
  Call Extruder(12.77611)
  MoveL 6290 to (-40.97, 148.02, 97.46) mm, rotated rx 180 ry 0 rz -180 deg; joints [-143.627, 67.07, -77.459, 143.174, 81.651, 6.205]
  MoveL 6291 to (-40.97, 148.02, 97.46) mm, rotated rx 180 ry 0 rz -180 deg; joints [-143.627, 67.07, -77.459, 143.174, 81.651, 6.205]
  Call Extruder(12.97282)
  MoveL 6292 to (-41.02, 147.63, 97.46) mm, rotated rx 180 ry 0 rz -180 deg; joints [-143.705, 67.058, -77.472, 143.25, 81.623, 6.209]
  MoveL 6293 to (-41.02, 147.63, 97.46) mm, rotated rx 180 ry 0 rz -180 deg; joints [-143.705, 67.058, -77.472, 143.25, 81.623, 6.209]
  Call Extruder(13.16866)
  MoveL 6294 to (-41.06, 147.25, 97.46) mm, rotated rx -180 ry 0 rz -180 deg; joints [-143.783, 67.047, -77.485, 143.326, 81.595, 6.212]
  MoveL 6295 to (-41.06, 147.25, 97.46) mm, rotated rx -180 ry 0 rz -180 deg; joints [-143.783, 67.047, -77.485, 143.326, 81.595, 6.212]
  Call Extruder(13.46406)
  MoveL 6296 to (-41.11, 146.66, 97.46) mm, rotated rx 180 ry 0 rz 180 deg; joints [-143.899, 67.028, -77.505, 143.439, 81.551, 6.219]
  MoveL 6297 to (-41.11, 146.66, 97.46) mm, rotated rx 180 ry 0 rz 180 deg; joints [-143.899, 67.028, -77.505, 143.439, 81.551, 6.219]
  Call Extruder(13.75812)
  MoveL 6298 to (-41.15, 146.07, 97.46) mm, rotated rx -180 ry 0 rz -180 deg; joints [-144.015, 67.009, -77.525, 143.552, 81.507, 6.225]
  MoveL 6299 to (-41.15, 146.07, 97.46) mm, rotated rx -180 ry 0 rz -180 deg; joints [-144.015, 67.009, -77.525, 143.552, 81.507, 6.225]
  Call Extruder(14.05086)
  MoveL 6300 to (-41.2, 145.48, 97.46) mm, rotated rx 180 ry 0 rz -180 deg; joints [-144.131, 66.99, -77.546, 143.666, 81.463, 6.231]
  MoveL 6301 to (-41.2, 145.48, 97.46) mm, rotated rx 180 ry 0 rz -180 deg; joints [-144.131, 66.99, -77.546, 143.666, 81.463, 6.231]
  Call Extruder(14.62431)
  MoveL 6302 to (-41.25, 144.32, 97.46) mm, rotated rx -180 ry 0 rz -180 deg; joints [-144.355, 66.95, -77.588, 143.884, 81.372, 6.246]
  MoveL 6303 to (-41.25, 144.32, 97.46) mm, rotated rx -180 ry 0 rz -180 deg; joints [-144.355, 66.95, -77.588, 143.884, 81.372, 6.246]
  Call Extruder(15.33827)
  MoveL 6304 to (-41.29, 142.86, 97.46) mm, rotated rx 180 ry 0 rz -180 deg; joints [-144.635, 66.9, -77.641, 144.156, 81.258, 6.265]
  Call Extruder(57.40309)
  MoveL 6305 to (-41.29, 57.14, 97.46) mm, rotated rx 180 ry 0 rz -180 deg; joints [-164.153, 64.346, -79.818, 163.588, 75.13, 4.323]
  Call Extruder(57.83164)
  MoveL 6306 to (-41.27, 56.26, 97.46) mm, rotated rx -180 ry 0 rz 180 deg; joints [-164.382, 64.327, -79.831, 163.823, 75.082, 4.271]
  MoveL 6307 to (-41.27, 56.26, 97.46) mm, rotated rx -180 ry 0 rz 180 deg; joints [-164.382, 64.327, -79.831, 163.823, 75.082, 4.271]
  Call Extruder(58.11773)
  MoveL 6308 to (-41.25, 55.68, 97.46) mm, rotated rx -180 ry 0 rz 180 deg; joints [-164.534, 64.314, -79.84, 163.978, 75.05, 4.237]
  MoveL 6309 to (-41.25, 55.68, 97.46) mm, rotated rx -180 ry 0 rz 180 deg; joints [-164.534, 64.314, -79.84, 163.978, 75.05, 4.237]
  Call Extruder(58.69247)
  MoveL 6310 to (-41.2, 54.52, 97.46) mm, rotated rx 180 ry 0 rz 180 deg; joints [-164.838, 64.288, -79.858, 164.289, 74.985, 4.168]
  MoveL 6311 to (-41.2, 54.52, 97.46) mm, rotated rx 180 ry 0 rz 180 deg; joints [-164.838, 64.288, -79.858, 164.289, 74.985, 4.168]
  Call Extruder(58.98586)
  MoveL 6312 to (-41.15, 53.93, 97.46) mm, rotated rx -180 ry 0 rz -180 deg; joints [-164.992, 64.273, -79.868, 164.445, 74.951, 4.134]
  MoveL 6313 to (-41.15, 53.93, 97.46) mm, rotated rx -180 ry 0 rz -180 deg; joints [-164.992, 64.273, -79.868, 164.445, 74.951, 4.134]
  Call Extruder(59.28059)
  MoveL 6314 to (-41.11, 53.34, 97.46) mm, rotated rx -180 ry 0 rz -180 deg; joints [-165.145, 64.259, -79.878, 164.602, 74.916, 4.099]
  MoveL 6315 to (-41.11, 53.34, 97.46) mm, rotated rx -180 ry 0 rz -180 deg; joints [-165.145, 64.259, -79.878, 164.602, 74.916, 4.099]
  Call Extruder(59.57665)
  MoveL 6316 to (-41.06, 52.75, 97.46) mm, rotated rx -180 ry 0 rz -180 deg; joints [-165.299, 64.244, -79.887, 164.759, 74.881, 4.065]
  MoveL 6317 to (-41.06, 52.75, 97.46) mm, rotated rx -180 ry 0 rz -180 deg; joints [-165.299, 64.244, -79.887, 164.759, 74.881, 4.065]
  Call Extruder(59.77292)
  MoveL 6318 to (-41.02, 52.36, 97.46) mm, rotated rx 180 ry 0 rz 180 deg; joints [-165.399, 64.234, -79.895, 164.861, 74.857, 4.042]
  MoveL 6319 to (-41.02, 52.36, 97.46) mm, rotated rx 180 ry 0 rz 180 deg; joints [-165.399, 64.234, -79.895, 164.861, 74.857, 4.042]
  Call Extruder(59.97006)
  MoveL 6320 to (-40.97, 51.98, 97.46) mm, rotated rx -180 ry 0 rz -180 deg; joints [-165.499, 64.223, -79.902, 164.964, 74.833, 4.02]
  MoveL 6321 to (-40.97, 51.98, 97.46) mm, rotated rx -180 ry 0 rz -180 deg; joints [-165.499, 64.223, -79.902, 164.964, 74.833, 4.02]
  Call Extruder(60.16807)
  MoveL 6322 to (-40.93, 51.59, 97.46) mm, rotated rx -180 ry 0 rz 180 deg; joints [-165.6, 64.213, -79.909, 165.066, 74.809, 3.998]
  MoveL 6323 to (-40.93, 51.59, 97.46) mm, rotated rx -180 ry 0 rz 180 deg; joints [-165.6, 64.213, -79.909, 165.066, 74.809, 3.998]
  Call Extruder(60.36695)
  MoveL 6324 to (-40.88, 51.2, 97.46) mm, rotated rx -180 ry 0 rz -180 deg; joints [-165.7, 64.202, -79.916, 165.169, 74.785, 3.975]
  MoveL 6325 to (-40.88, 51.2, 97.46) mm, rotated rx -180 ry 0 rz -180 deg; joints [-165.7, 64.202, -79.916, 165.169, 74.785, 3.975]
  Call Extruder(60.54602)
  MoveL 6326 to (-40.83, 50.86, 97.46) mm, rotated rx 180 ry 0 rz -180 deg; joints [-165.79, 64.193, -79.922, 165.261, 74.763, 3.955]
  MoveL 6327 to (-40.83, 50.86, 97.46) mm, rotated rx 180 ry 0 rz -180 deg; joints [-165.79, 64.193, -79.922, 165.261, 74.763, 3.955]
  Call Extruder(60.70520)
  MoveL 6328 to (-40.78, 50.55, 97.46) mm, rotated rx -180 ry 0 rz -180 deg; joints [-165.869, 64.184, -79.928, 165.341, 74.743, 3.938]
  MoveL 6329 to (-40.78, 50.55, 97.46) mm, rotated rx -180 ry 0 rz -180 deg; joints [-165.869, 64.184, -79.928, 165.341, 74.743, 3.938]
  Call Extruder(60.86511)
  MoveL 6330 to (-40.74, 50.24, 97.46) mm, rotated rx -180 ry 0 rz 180 deg; joints [-165.948, 64.175, -79.935, 165.422, 74.723, 3.92]
  MoveL 6331 to (-40.74, 50.24, 97.46) mm, rotated rx -180 ry 0 rz 180 deg; joints [-165.948, 64.175, -79.935, 165.422, 74.723, 3.92]
  Call Extruder(61.02575)
  MoveL 6332 to (-40.69, 49.94, 97.46) mm, rotated rx -180 ry 0 rz -180 deg; joints [-166.026, 64.165, -79.941, 165.502, 74.703, 3.903]
  MoveL 6333 to (-40.69, 49.94, 97.46) mm, rotated rx -180 ry 0 rz -180 deg; joints [-166.026, 64.165, -79.941, 165.502, 74.703, 3.903]
  Call Extruder(61.18711)
  MoveL 6334 to (-40.64, 49.63, 97.46) mm, rotated rx -180 ry 0 rz -180 deg; joints [-166.105, 64.156, -79.947, 165.583, 74.683, 3.885]
  MoveL 6335 to (-40.64, 49.63, 97.46) mm, rotated rx -180 ry 0 rz -180 deg; joints [-166.105, 64.156, -79.947, 165.583, 74.683, 3.885]
  Call Extruder(61.34921)
  MoveL 6336 to (-40.59, 49.33, 97.46) mm, rotated rx -180 ry 0 rz -180 deg; joints [-166.184, 64.147, -79.953, 165.664, 74.664, 3.867]
  MoveL 6337 to (-40.59, 49.33, 97.46) mm, rotated rx -180 ry 0 rz -180 deg; joints [-166.184, 64.147, -79.953, 165.664, 74.664, 3.867]
  Call Extruder(61.49740)
  MoveL 6338 to (-40.54, 49.05, 97.46) mm, rotated rx -180 ry 0 rz -180 deg; joints [-166.256, 64.139, -79.958, 165.737, 74.645, 3.851]
  MoveL 6339 to (-40.54, 49.05, 97.46) mm, rotated rx -180 ry 0 rz -180 deg; joints [-166.256, 64.139, -79.958, 165.737, 74.645, 3.851]
  Call Extruder(61.63163)
  MoveL 6340 to (-40.49, 48.8, 97.46) mm, rotated rx 180 ry 0 rz 180 deg; joints [-166.32, 64.131, -79.964, 165.802, 74.628, 3.837]
  MoveL 6341 to (-40.49, 48.8, 97.46) mm, rotated rx 180 ry 0 rz 180 deg; joints [-166.32, 64.131, -79.964, 165.802, 74.628, 3.837]
  Call Extruder(61.76647)
  MoveL 6342 to (-40.44, 48.55, 97.46) mm, rotated rx -180 ry 0 rz -180 deg; joints [-166.384, 64.123, -79.969, 165.867, 74.611, 3.823]
  MoveL 6343 to (-40.44, 48.55, 97.46) mm, rotated rx -180 ry 0 rz -180 deg; joints [-166.384, 64.123, -79.969, 165.867, 74.611, 3.823]
  Call Extruder(61.90192)
  MoveL 6344 to (-40.39, 48.3, 97.46) mm, rotated rx -180 ry 0 rz 180 deg; joints [-166.448, 64.115, -79.974, 165.932, 74.594, 3.809]
  MoveL 6345 to (-40.39, 48.3, 97.46) mm, rotated rx -180 ry 0 rz 180 deg; joints [-166.448, 64.115, -79.974, 165.932, 74.594, 3.809]
  Call Extruder(62.03798)
  MoveL 6346 to (-40.34, 48.05, 97.46) mm, rotated rx -180 ry 0 rz -180 deg; joints [-166.512, 64.107, -79.979, 165.998, 74.577, 3.794]
  MoveL 6347 to (-40.34, 48.05, 97.46) mm, rotated rx -180 ry 0 rz -180 deg; joints [-166.512, 64.107, -79.979, 165.998, 74.577, 3.794]
  Call Extruder(62.17465)
  MoveL 6348 to (-40.29, 47.8, 97.46) mm, rotated rx -180 ry 0 rz 180 deg; joints [-166.576, 64.099, -79.985, 166.064, 74.559, 3.78]
  MoveL 6349 to (-40.29, 47.8, 97.46) mm, rotated rx -180 ry 0 rz 180 deg; joints [-166.576, 64.099, -79.985, 166.064, 74.559, 3.78]
  Call Extruder(62.31193)
  MoveL 6350 to (-40.24, 47.56, 97.46) mm, rotated rx -180 ry 0 rz 180 deg; joints [-166.641, 64.091, -79.99, 166.129, 74.542, 3.765]
  MoveL 6351 to (-40.24, 47.56, 97.46) mm, rotated rx -180 ry 0 rz 180 deg; joints [-166.641, 64.091, -79.99, 166.129, 74.542, 3.765]
  Call Extruder(62.43761)
  MoveL 6352 to (-40.2, 47.33, 97.46) mm, rotated rx -180 ry 0 rz -180 deg; joints [-166.699, 64.084, -79.995, 166.189, 74.527, 3.752]
  MoveL 6353 to (-40.2, 47.33, 97.46) mm, rotated rx -180 ry 0 rz -180 deg; joints [-166.699, 64.084, -79.995, 166.189, 74.527, 3.752]
  Call Extruder(62.55156)
  MoveL 6354 to (-40.15, 47.12, 97.46) mm, rotated rx -180 ry 0 rz 180 deg; joints [-166.751, 64.077, -79.999, 166.243, 74.512, 3.741]
  MoveL 6355 to (-40.15, 47.12, 97.46) mm, rotated rx -180 ry 0 rz 180 deg; joints [-166.751, 64.077, -79.999, 166.243, 74.512, 3.741]
  Call Extruder(62.66597)
  MoveL 6356 to (-40.11, 46.92, 97.46) mm, rotated rx -180 ry 0 rz -180 deg; joints [-166.804, 64.07, -80.004, 166.296, 74.498, 3.729]
  MoveL 6357 to (-40.11, 46.92, 97.46) mm, rotated rx -180 ry 0 rz -180 deg; joints [-166.804, 64.07, -80.004, 166.296, 74.498, 3.729]
  Call Extruder(62.78083)
  MoveL 6358 to (-40.06, 46.72, 97.46) mm, rotated rx 180 ry 0 rz -180 deg; joints [-166.857, 64.064, -80.008, 166.35, 74.484, 3.717]
  MoveL 6359 to (-40.06, 46.72, 97.46) mm, rotated rx 180 ry 0 rz -180 deg; joints [-166.857, 64.064, -80.008, 166.35, 74.484, 3.717]
  Call Extruder(62.89614)
  MoveL 6360 to (-40.02, 46.51, 97.46) mm, rotated rx -180 ry 0 rz -180 deg; joints [-166.909, 64.057, -80.013, 166.404, 74.47, 3.705]
  MoveL 6361 to (-40.02, 46.51, 97.46) mm, rotated rx -180 ry 0 rz -180 deg; joints [-166.909, 64.057, -80.013, 166.404, 74.47, 3.705]
  Call Extruder(63.02552)
  MoveL 6362 to (-39.95, 46.29, 97.46) mm, rotated rx -180 ry 0 rz 180 deg; joints [-166.966, 64.048, -80.018, 166.461, 74.452, 3.693]
  MoveL 6363 to (-39.95, 46.29, 97.46) mm, rotated rx -180 ry 0 rz 180 deg; joints [-166.966, 64.048, -80.018, 166.461, 74.452, 3.693]
  Call Extruder(63.15547)
  MoveL 6364 to (-39.88, 46.06, 97.46) mm, rotated rx 180 ry 0 rz 180 deg; joints [-167.022, 64.04, -80.024, 166.519, 74.434, 3.681]
  MoveL 6365 to (-39.88, 46.06, 97.46) mm, rotated rx 180 ry 0 rz 180 deg; joints [-167.022, 64.04, -80.024, 166.519, 74.434, 3.681]
  Call Extruder(63.28598)
  MoveL 6366 to (-39.81, 45.84, 97.46) mm, rotated rx -180 ry 0 rz -180 deg; joints [-167.079, 64.031, -80.03, 166.577, 74.417, 3.668]
  MoveL 6367 to (-39.81, 45.84, 97.46) mm, rotated rx -180 ry 0 rz -180 deg; joints [-167.079, 64.031, -80.03, 166.577, 74.417, 3.668]
  Call Extruder(63.41705)
  MoveL 6368 to (-39.75, 45.62, 97.46) mm, rotated rx -180 ry 0 rz -180 deg; joints [-167.136, 64.022, -80.036, 166.635, 74.399, 3.656]
  MoveL 6369 to (-39.75, 45.62, 97.46) mm, rotated rx -180 ry 0 rz -180 deg; joints [-167.136, 64.022, -80.036, 166.635, 74.399, 3.656]
  Call Extruder(63.53870)
  MoveL 6370 to (-39.68, 45.41, 97.46) mm, rotated rx 180 ry 0 rz -180 deg; joints [-167.188, 64.014, -80.041, 166.688, 74.382, 3.645]
  MoveL 6371 to (-39.68, 45.41, 97.46) mm, rotated rx 180 ry 0 rz -180 deg; joints [-167.188, 64.014, -80.041, 166.688, 74.382, 3.645]
  Call Extruder(63.65082)
  MoveL 6372 to (-39.62, 45.22, 97.46) mm, rotated rx -180 ry 0 rz -180 deg; joints [-167.235, 64.006, -80.046, 166.736, 74.367, 3.635]
  MoveL 6373 to (-39.62, 45.22, 97.46) mm, rotated rx -180 ry 0 rz -180 deg; joints [-167.235, 64.006, -80.046, 166.736, 74.367, 3.635]
  Call Extruder(63.76339)
  MoveL 6374 to (-39.56, 45.03, 97.46) mm, rotated rx 180 ry 0 rz -180 deg; joints [-167.283, 63.999, -80.051, 166.785, 74.352, 3.624]
  MoveL 6375 to (-39.56, 45.03, 97.46) mm, rotated rx 180 ry 0 rz -180 deg; joints [-167.283, 63.999, -80.051, 166.785, 74.352, 3.624]
  Call Extruder(63.87640)
  MoveL 6376 to (-39.5, 44.85, 97.46) mm, rotated rx -180 ry 0 rz 180 deg; joints [-167.331, 63.991, -80.056, 166.834, 74.337, 3.614]
  MoveL 6377 to (-39.5, 44.85, 97.46) mm, rotated rx -180 ry 0 rz 180 deg; joints [-167.331, 63.991, -80.056, 166.834, 74.337, 3.614]
  Call Extruder(63.98986)
  MoveL 6378 to (-39.44, 44.66, 97.46) mm, rotated rx -180 ry 0 rz 180 deg; joints [-167.379, 63.983, -80.061, 166.882, 74.321, 3.603]
  MoveL 6379 to (-39.44, 44.66, 97.46) mm, rotated rx -180 ry 0 rz 180 deg; joints [-167.379, 63.983, -80.061, 166.882, 74.321, 3.603]
  Call Extruder(64.13750)
  MoveL 6380 to (-39.35, 44.42, 97.46) mm, rotated rx 180 ry 0 rz 180 deg; joints [-167.439, 63.973, -80.068, 166.944, 74.3, 3.591]
  MoveL 6381 to (-39.35, 44.42, 97.46) mm, rotated rx 180 ry 0 rz 180 deg; joints [-167.439, 63.973, -80.068, 166.944, 74.3, 3.591]
  Call Extruder(64.31984)
  MoveL 6382 to (-39.23, 44.12, 97.46) mm, rotated rx 180 ry 0 rz 180 deg; joints [-167.512, 63.959, -80.077, 167.018, 74.274, 3.576]
  MoveL 6383 to (-39.23, 44.12, 97.46) mm, rotated rx 180 ry 0 rz 180 deg; joints [-167.512, 63.959, -80.077, 167.018, 74.274, 3.576]
  Call Extruder(64.50294)
  MoveL 6384 to (-39.11, 43.83, 97.46) mm, rotated rx 180 ry 0 rz -180 deg; joints [-167.584, 63.946, -80.085, 167.092, 74.248, 3.56]
  MoveL 6385 to (-39.11, 43.83, 97.46) mm, rotated rx 180 ry 0 rz -180 deg; joints [-167.584, 63.946, -80.085, 167.092, 74.248, 3.56]
  Call Extruder(64.66062)
  MoveL 6386 to (-39, 43.58, 97.46) mm, rotated rx 180 ry 0 rz 180 deg; joints [-167.646, 63.934, -80.093, 167.155, 74.225, 3.547]
  MoveL 6387 to (-39, 43.58, 97.46) mm, rotated rx 180 ry 0 rz 180 deg; joints [-167.646, 63.934, -80.093, 167.155, 74.225, 3.547]
  Call Extruder(64.81891)
  MoveL 6388 to (-38.89, 43.33, 97.46) mm, rotated rx -180 ry 0 rz 180 deg; joints [-167.708, 63.922, -80.101, 167.218, 74.202, 3.534]
  MoveL 6389 to (-38.89, 43.33, 97.46) mm, rotated rx -180 ry 0 rz 180 deg; joints [-167.708, 63.922, -80.101, 167.218, 74.202, 3.534]
  Call Extruder(65.00093)
  MoveL 6390 to (-38.75, 43.06, 97.46) mm, rotated rx 180 ry 0 rz -180 deg; joints [-167.776, 63.907, -80.11, 167.287, 74.174, 3.521]
  MoveL 6391 to (-38.75, 43.06, 97.46) mm, rotated rx 180 ry 0 rz -180 deg; joints [-167.776, 63.907, -80.11, 167.287, 74.174, 3.521]
  Call Extruder(65.20748)
  MoveL 6392 to (-38.57, 42.75, 97.46) mm, rotated rx -180 ry 0 rz -180 deg; joints [-167.849, 63.889, -80.122, 167.361, 74.141, 3.507]
  MoveL 6393 to (-38.57, 42.75, 97.46) mm, rotated rx -180 ry 0 rz -180 deg; joints [-167.849, 63.889, -80.122, 167.361, 74.141, 3.507]
  Call Extruder(65.41481)
  MoveL 6394 to (-38.4, 42.45, 97.46) mm, rotated rx -180 ry 0 rz 180 deg; joints [-167.923, 63.871, -80.133, 167.435, 74.108, 3.492]
  MoveL 6395 to (-38.4, 42.45, 97.46) mm, rotated rx -180 ry 0 rz 180 deg; joints [-167.923, 63.871, -80.133, 167.435, 74.108, 3.492]
  Call Extruder(65.62293)
  MoveL 6396 to (-38.22, 42.15, 97.46) mm, rotated rx -180 ry 0 rz -180 deg; joints [-167.997, 63.854, -80.145, 167.51, 74.075, 3.478]
  MoveL 6397 to (-38.22, 42.15, 97.46) mm, rotated rx -180 ry 0 rz -180 deg; joints [-167.997, 63.854, -80.145, 167.51, 74.075, 3.478]
  Call Extruder(65.74064)
  MoveL 6398 to (-38.12, 41.98, 97.46) mm, rotated rx 180 ry 0 rz 180 deg; joints [-168.038, 63.843, -80.151, 167.552, 74.056, 3.47]
  MoveL 6399 to (-38.12, 41.98, 97.46) mm, rotated rx 180 ry 0 rz 180 deg; joints [-168.038, 63.843, -80.151, 167.552, 74.056, 3.47]
  Call Extruder(66.07349)
  MoveL 6400 to (-37.8, 41.52, 97.46) mm, rotated rx -180 ry 0 rz -180 deg; joints [-168.144, 63.812, -80.171, 167.659, 73.999, 3.451]
  MoveL 6401 to (-37.8, 41.52, 97.46) mm, rotated rx -180 ry 0 rz -180 deg; joints [-168.144, 63.812, -80.171, 167.659, 73.999, 3.451]
  Call Extruder(66.40752)
  MoveL 6402 to (-37.47, 41.07, 97.46) mm, rotated rx -180 ry 0 rz -180 deg; joints [-168.25, 63.781, -80.191, 167.766, 73.943, 3.432]
  MoveL 6403 to (-37.47, 41.07, 97.46) mm, rotated rx -180 ry 0 rz -180 deg; joints [-168.25, 63.781, -80.191, 167.766, 73.943, 3.432]
  Call Extruder(66.57511)
  MoveL 6404 to (-37.3, 40.85, 97.46) mm, rotated rx 180 ry 0 rz -180 deg; joints [-168.304, 63.765, -80.201, 167.82, 73.915, 3.422]
  Call Extruder(67.40442)
  MoveL 6405 to (-36.39, 39.81, 97.46) mm, rotated rx 180 ry 0 rz 180 deg; joints [-168.541, 63.681, -80.253, 168.059, 73.767, 3.383]
  Call Extruder(68.03549)
  MoveL 6406 to (-35.61, 39.11, 97.46) mm, rotated rx -180 ry 0 rz 180 deg; joints [-168.693, 63.611, -80.296, 168.21, 73.648, 3.363]
  MoveL 6407 to (-35.61, 39.11, 97.46) mm, rotated rx -180 ry 0 rz 180 deg; joints [-168.693, 63.611, -80.296, 168.21, 73.648, 3.363]
  Call Extruder(68.23306)
  MoveL 6408 to (-35.35, 38.9, 97.46) mm, rotated rx 180 ry 0 rz 180 deg; joints [-168.739, 63.589, -80.31, 168.255, 73.61, 3.357]
  Call Extruder(68.56708)
  MoveL 6409 to (-34.9, 38.57, 97.46) mm, rotated rx 180 ry 0 rz -180 deg; joints [-168.806, 63.55, -80.334, 168.322, 73.545, 3.351]
  MoveL 6410 to (-34.9, 38.57, 97.46) mm, rotated rx 180 ry 0 rz -180 deg; joints [-168.806, 63.55, -80.334, 168.322, 73.545, 3.351]
  Call Extruder(68.89991)
  MoveL 6411 to (-34.45, 38.24, 97.46) mm, rotated rx 180 ry 0 rz 180 deg; joints [-168.874, 63.511, -80.357, 168.389, 73.48, 3.344]
  MoveL 6412 to (-34.45, 38.24, 97.46) mm, rotated rx 180 ry 0 rz 180 deg; joints [-168.874, 63.511, -80.357, 168.389, 73.48, 3.344]
  Call Extruder(69.07916)
  MoveL 6413 to (-34.21, 38.07, 97.46) mm, rotated rx 180 ry 0 rz -180 deg; joints [-168.91, 63.49, -80.37, 168.424, 73.444, 3.34]
  MoveL 6414 to (-34.21, 38.07, 97.46) mm, rotated rx 180 ry 0 rz -180 deg; joints [-168.91, 63.49, -80.37, 168.424, 73.444, 3.34]
  Call Extruder(69.28727)
  MoveL 6415 to (-33.9, 37.89, 97.46) mm, rotated rx -180 ry 0 rz 180 deg; joints [-168.944, 63.464, -80.386, 168.456, 73.402, 3.339]
  MoveL 6416 to (-33.9, 37.89, 97.46) mm, rotated rx -180 ry 0 rz 180 deg; joints [-168.944, 63.464, -80.386, 168.456, 73.402, 3.339]
  Call Extruder(69.49460)
  MoveL 6417 to (-33.6, 37.71, 97.46) mm, rotated rx 180 ry 0 rz 180 deg; joints [-168.977, 63.439, -80.401, 168.488, 73.36, 3.338]
  MoveL 6418 to (-33.6, 37.71, 97.46) mm, rotated rx 180 ry 0 rz 180 deg; joints [-168.977, 63.439, -80.401, 168.488, 73.36, 3.338]
  Call Extruder(69.70115)
  MoveL 6419 to (-33.29, 37.54, 97.46) mm, rotated rx 180 ry 0 rz -180 deg; joints [-169.01, 63.413, -80.416, 168.521, 73.318, 3.336]
  MoveL 6420 to (-33.29, 37.54, 97.46) mm, rotated rx 180 ry 0 rz -180 deg; joints [-169.01, 63.413, -80.416, 168.521, 73.318, 3.336]
  Call Extruder(69.90692)
  MoveL 6421 to (-32.99, 37.36, 97.46) mm, rotated rx 180 ry 0 rz -180 deg; joints [-169.043, 63.387, -80.432, 168.553, 73.276, 3.335]
  MoveL 6422 to (-32.99, 37.36, 97.46) mm, rotated rx 180 ry 0 rz -180 deg; joints [-169.043, 63.387, -80.432, 168.553, 73.276, 3.335]
  Call Extruder(70.06522)
  MoveL 6423 to (-32.74, 37.26, 97.46) mm, rotated rx 180 ry 0 rz 180 deg; joints [-169.06, 63.367, -80.444, 168.568, 73.243, 3.337]
  MoveL 6424 to (-32.74, 37.26, 97.46) mm, rotated rx 180 ry 0 rz 180 deg; joints [-169.06, 63.367, -80.444, 168.568, 73.243, 3.337]
  Call Extruder(70.22292)
  MoveL 6425 to (-32.49, 37.15, 97.46) mm, rotated rx -180 ry 0 rz -180 deg; joints [-169.077, 63.346, -80.456, 168.584, 73.209, 3.338]
  MoveL 6426 to (-32.49, 37.15, 97.46) mm, rotated rx -180 ry 0 rz -180 deg; joints [-169.077, 63.346, -80.456, 168.584, 73.209, 3.338]
  Call Extruder(70.39301)
  MoveL 6427 to (-32.22, 37.03, 97.46) mm, rotated rx -180 ry 0 rz 180 deg; joints [-169.095, 63.324, -80.469, 168.6, 73.174, 3.34]
  MoveL 6428 to (-32.22, 37.03, 97.46) mm, rotated rx -180 ry 0 rz 180 deg; joints [-169.095, 63.324, -80.469, 168.6, 73.174, 3.34]
  Call Extruder(70.57534)
  MoveL 6429 to (-31.93, 36.91, 97.46) mm, rotated rx 180 ry 0 rz 180 deg; joints [-169.113, 63.3, -80.483, 168.617, 73.135, 3.343]
  MoveL 6430 to (-31.93, 36.91, 97.46) mm, rotated rx 180 ry 0 rz 180 deg; joints [-169.113, 63.3, -80.483, 168.617, 73.135, 3.343]
  Call Extruder(70.75692)
  MoveL 6431 to (-31.64, 36.79, 97.46) mm, rotated rx -180 ry 0 rz 180 deg; joints [-169.132, 63.276, -80.497, 168.635, 73.097, 3.345]
  MoveL 6432 to (-31.64, 36.79, 97.46) mm, rotated rx -180 ry 0 rz 180 deg; joints [-169.132, 63.276, -80.497, 168.635, 73.097, 3.345]
  Call Extruder(70.87038)
  MoveL 6433 to (-31.45, 36.73, 97.46) mm, rotated rx -180 ry 0 rz 180 deg; joints [-169.139, 63.26, -80.506, 168.641, 73.072, 3.348]
  MoveL 6434 to (-31.45, 36.73, 97.46) mm, rotated rx -180 ry 0 rz 180 deg; joints [-169.139, 63.26, -80.506, 168.641, 73.072, 3.348]
  Call Extruder(70.98339)
  MoveL 6435 to (-31.26, 36.67, 97.46) mm, rotated rx -180 ry 0 rz -180 deg; joints [-169.146, 63.245, -80.515, 168.647, 73.048, 3.35]
  MoveL 6436 to (-31.26, 36.67, 97.46) mm, rotated rx -180 ry 0 rz -180 deg; joints [-169.146, 63.245, -80.515, 168.647, 73.048, 3.35]
  Call Extruder(71.09596)
  MoveL 6437 to (-31.07, 36.61, 97.46) mm, rotated rx -180 ry 0 rz -180 deg; joints [-169.154, 63.23, -80.524, 168.653, 73.024, 3.353]
  MoveL 6438 to (-31.07, 36.61, 97.46) mm, rotated rx -180 ry 0 rz -180 deg; joints [-169.154, 63.23, -80.524, 168.653, 73.024, 3.353]
  Call Extruder(71.20808)
  MoveL 6439 to (-30.88, 36.55, 97.46) mm, rotated rx -180 ry 0 rz 180 deg; joints [-169.161, 63.214, -80.533, 168.659, 73, 3.356]
  MoveL 6440 to (-30.88, 36.55, 97.46) mm, rotated rx -180 ry 0 rz 180 deg; joints [-169.161, 63.214, -80.533, 168.659, 73, 3.356]
  Call Extruder(71.31976)
  MoveL 6441 to (-30.7, 36.49, 97.46) mm, rotated rx -180 ry 0 rz 180 deg; joints [-169.168, 63.199, -80.542, 168.665, 72.975, 3.359]
  MoveL 6442 to (-30.7, 36.49, 97.46) mm, rotated rx -180 ry 0 rz 180 deg; joints [-169.168, 63.199, -80.542, 168.665, 72.975, 3.359]
  Call Extruder(71.45084)
  MoveL 6443 to (-30.47, 36.42, 97.46) mm, rotated rx -180 ry 0 rz 180 deg; joints [-169.175, 63.181, -80.552, 168.671, 72.947, 3.362]
  MoveL 6444 to (-30.47, 36.42, 97.46) mm, rotated rx -180 ry 0 rz 180 deg; joints [-169.175, 63.181, -80.552, 168.671, 72.947, 3.362]
  Call Extruder(71.58135)
  MoveL 6445 to (-30.25, 36.35, 97.46) mm, rotated rx -180 ry 0 rz 180 deg; joints [-169.182, 63.162, -80.563, 168.677, 72.918, 3.366]
  MoveL 6446 to (-30.25, 36.35, 97.46) mm, rotated rx -180 ry 0 rz 180 deg; joints [-169.182, 63.162, -80.563, 168.677, 72.918, 3.366]
  Call Extruder(71.71129)
  MoveL 6447 to (-30.02, 36.28, 97.46) mm, rotated rx 180 ry 0 rz -180 deg; joints [-169.19, 63.144, -80.573, 168.683, 72.89, 3.37]
  MoveL 6448 to (-30.02, 36.28, 97.46) mm, rotated rx 180 ry 0 rz -180 deg; joints [-169.19, 63.144, -80.573, 168.683, 72.89, 3.37]
  Call Extruder(71.84067)
  MoveL 6449 to (-29.8, 36.22, 97.46) mm, rotated rx -180 ry 0 rz -180 deg; joints [-169.197, 63.126, -80.584, 168.689, 72.861, 3.373]
  MoveL 6450 to (-29.8, 36.22, 97.46) mm, rotated rx -180 ry 0 rz -180 deg; joints [-169.197, 63.126, -80.584, 168.689, 72.861, 3.373]
  Call Extruder(71.96263)
  MoveL 6451 to (-29.59, 36.16, 97.46) mm, rotated rx -180 ry 0 rz -180 deg; joints [-169.202, 63.109, -80.594, 168.692, 72.834, 3.378]
  MoveL 6452 to (-29.59, 36.16, 97.46) mm, rotated rx -180 ry 0 rz -180 deg; joints [-169.202, 63.109, -80.594, 168.692, 72.834, 3.378]
  Call Extruder(72.07748)
  MoveL 6453 to (-29.38, 36.12, 97.46) mm, rotated rx -180 ry 0 rz 180 deg; joints [-169.203, 63.092, -80.603, 168.692, 72.809, 3.382]
  MoveL 6454 to (-29.38, 36.12, 97.46) mm, rotated rx -180 ry 0 rz 180 deg; joints [-169.203, 63.092, -80.603, 168.692, 72.809, 3.382]
  Call Extruder(72.19188)
  MoveL 6455 to (-29.18, 36.07, 97.46) mm, rotated rx -180 ry 0 rz -180 deg; joints [-169.205, 63.076, -80.612, 168.692, 72.784, 3.387]
  MoveL 6456 to (-29.18, 36.07, 97.46) mm, rotated rx -180 ry 0 rz -180 deg; joints [-169.205, 63.076, -80.612, 168.692, 72.784, 3.387]
  Call Extruder(72.30582)
  MoveL 6457 to (-28.97, 36.03, 97.46) mm, rotated rx 180 ry 0 rz -180 deg; joints [-169.207, 63.059, -80.622, 168.692, 72.758, 3.392]
  MoveL 6458 to (-28.97, 36.03, 97.46) mm, rotated rx 180 ry 0 rz -180 deg; joints [-169.207, 63.059, -80.622, 168.692, 72.758, 3.392]
  Call Extruder(72.41931)
  MoveL 6459 to (-28.77, 35.98, 97.46) mm, rotated rx -180 ry 0 rz -180 deg; joints [-169.208, 63.043, -80.631, 168.692, 72.733, 3.397]
  MoveL 6460 to (-28.77, 35.98, 97.46) mm, rotated rx -180 ry 0 rz -180 deg; joints [-169.208, 63.043, -80.631, 168.692, 72.733, 3.397]
  Call Extruder(72.55660)
  MoveL 6461 to (-28.52, 35.93, 97.46) mm, rotated rx 180 ry 0 rz 180 deg; joints [-169.209, 63.023, -80.642, 168.691, 72.702, 3.403]
  MoveL 6462 to (-28.52, 35.93, 97.46) mm, rotated rx 180 ry 0 rz 180 deg; joints [-169.209, 63.023, -80.642, 168.691, 72.702, 3.403]
  Call Extruder(72.69327)
  MoveL 6463 to (-28.27, 35.88, 97.46) mm, rotated rx -180 ry 0 rz -180 deg; joints [-169.209, 63.003, -80.653, 168.69, 72.671, 3.409]
  MoveL 6464 to (-28.27, 35.88, 97.46) mm, rotated rx -180 ry 0 rz -180 deg; joints [-169.209, 63.003, -80.653, 168.69, 72.671, 3.409]
  Call Extruder(72.82933)
  MoveL 6465 to (-28.02, 35.83, 97.46) mm, rotated rx -180 ry 0 rz 180 deg; joints [-169.21, 62.983, -80.665, 168.688, 72.641, 3.415]
  MoveL 6466 to (-28.02, 35.83, 97.46) mm, rotated rx -180 ry 0 rz 180 deg; joints [-169.21, 62.983, -80.665, 168.688, 72.641, 3.415]
  Call Extruder(72.96478)
  MoveL 6467 to (-27.77, 35.78, 97.46) mm, rotated rx -180 ry 0 rz -180 deg; joints [-169.21, 62.962, -80.676, 168.687, 72.61, 3.422]
  MoveL 6468 to (-27.77, 35.78, 97.46) mm, rotated rx -180 ry 0 rz -180 deg; joints [-169.21, 62.962, -80.676, 168.687, 72.61, 3.422]
  Call Extruder(73.09962)
  MoveL 6469 to (-27.52, 35.73, 97.46) mm, rotated rx -180 ry 0 rz 180 deg; joints [-169.211, 62.942, -80.687, 168.686, 72.579, 3.428]
  MoveL 6470 to (-27.52, 35.73, 97.46) mm, rotated rx -180 ry 0 rz 180 deg; joints [-169.211, 62.942, -80.687, 168.686, 72.579, 3.428]
  Call Extruder(73.23385)
  MoveL 6471 to (-27.28, 35.68, 97.46) mm, rotated rx 180 ry 0 rz 180 deg; joints [-169.212, 62.922, -80.698, 168.685, 72.548, 3.434]
  MoveL 6472 to (-27.28, 35.68, 97.46) mm, rotated rx 180 ry 0 rz 180 deg; joints [-169.212, 62.922, -80.698, 168.685, 72.548, 3.434]
  Call Extruder(73.36747)
  MoveL 6473 to (-27.03, 35.63, 97.46) mm, rotated rx -180 ry 0 rz -180 deg; joints [-169.212, 62.902, -80.709, 168.683, 72.518, 3.44]
  MoveL 6474 to (-27.03, 35.63, 97.46) mm, rotated rx -180 ry 0 rz -180 deg; joints [-169.212, 62.902, -80.709, 168.683, 72.518, 3.44]
  Call Extruder(73.52957)
  MoveL 6475 to (-26.72, 35.59, 97.46) mm, rotated rx 180 ry 0 rz 180 deg; joints [-169.21, 62.877, -80.723, 168.678, 72.481, 3.449]
  MoveL 6476 to (-26.72, 35.59, 97.46) mm, rotated rx 180 ry 0 rz 180 deg; joints [-169.21, 62.877, -80.723, 168.678, 72.481, 3.449]
  Call Extruder(73.69094)
  MoveL 6477 to (-26.41, 35.54, 97.46) mm, rotated rx -180 ry 0 rz -180 deg; joints [-169.207, 62.853, -80.736, 168.672, 72.443, 3.458]
  MoveL 6478 to (-26.41, 35.54, 97.46) mm, rotated rx -180 ry 0 rz -180 deg; joints [-169.207, 62.853, -80.736, 168.672, 72.443, 3.458]
  Call Extruder(73.85158)
  MoveL 6479 to (-26.11, 35.49, 97.46) mm, rotated rx -180 ry 0 rz -180 deg; joints [-169.204, 62.828, -80.75, 168.667, 72.406, 3.467]
  MoveL 6480 to (-26.11, 35.49, 97.46) mm, rotated rx -180 ry 0 rz -180 deg; joints [-169.204, 62.828, -80.75, 168.667, 72.406, 3.467]
  Call Extruder(74.01150)
  MoveL 6481 to (-25.8, 35.44, 97.46) mm, rotated rx -180 ry 0 rz 180 deg; joints [-169.201, 62.804, -80.763, 168.662, 72.369, 3.475]
  MoveL 6482 to (-25.8, 35.44, 97.46) mm, rotated rx -180 ry 0 rz 180 deg; joints [-169.201, 62.804, -80.763, 168.662, 72.369, 3.475]
  Call Extruder(74.17068)
  MoveL 6483 to (-25.5, 35.39, 97.46) mm, rotated rx 180 ry 0 rz 180 deg; joints [-169.198, 62.779, -80.776, 168.656, 72.332, 3.484]
  MoveL 6484 to (-25.5, 35.39, 97.46) mm, rotated rx 180 ry 0 rz 180 deg; joints [-169.198, 62.779, -80.776, 168.656, 72.332, 3.484]
  Call Extruder(74.32914)
  MoveL 6485 to (-25.19, 35.34, 97.46) mm, rotated rx 180 ry 0 rz -180 deg; joints [-169.195, 62.754, -80.79, 168.651, 72.295, 3.493]
  MoveL 6486 to (-25.19, 35.34, 97.46) mm, rotated rx 180 ry 0 rz -180 deg; joints [-169.195, 62.754, -80.79, 168.651, 72.295, 3.493]
  Call Extruder(74.52802)
  MoveL 6487 to (-24.8, 35.3, 97.46) mm, rotated rx -180 ry 0 rz -180 deg; joints [-169.187, 62.723, -80.806, 168.639, 72.248, 3.506]
  MoveL 6488 to (-24.8, 35.3, 97.46) mm, rotated rx -180 ry 0 rz -180 deg; joints [-169.187, 62.723, -80.806, 168.639, 72.248, 3.506]
  Call Extruder(74.72603)
  MoveL 6489 to (-24.42, 35.25, 97.46) mm, rotated rx -180 ry 0 rz -180 deg; joints [-169.178, 62.692, -80.823, 168.627, 72.202, 3.518]
  MoveL 6490 to (-24.42, 35.25, 97.46) mm, rotated rx -180 ry 0 rz -180 deg; joints [-169.178, 62.692, -80.823, 168.627, 72.202, 3.518]
  Call Extruder(74.92317)
  MoveL 6491 to (-24.03, 35.21, 97.46) mm, rotated rx -180 ry 0 rz -180 deg; joints [-169.17, 62.661, -80.84, 168.615, 72.156, 3.531]
  MoveL 6492 to (-24.03, 35.21, 97.46) mm, rotated rx -180 ry 0 rz -180 deg; joints [-169.17, 62.661, -80.84, 168.615, 72.156, 3.531]
  Call Extruder(75.11944)
  MoveL 6493 to (-23.64, 35.16, 97.46) mm, rotated rx -180 ry 0 rz 180 deg; joints [-169.161, 62.629, -80.856, 168.603, 72.109, 3.543]
  MoveL 6494 to (-23.64, 35.16, 97.46) mm, rotated rx -180 ry 0 rz 180 deg; joints [-169.161, 62.629, -80.856, 168.603, 72.109, 3.543]
  Call Extruder(75.36513)
  MoveL 6495 to (-23.15, 35.11, 97.46) mm, rotated rx -180 ry 0 rz 180 deg; joints [-169.147, 62.59, -80.877, 168.584, 72.051, 3.561]
  MoveL 6496 to (-23.15, 35.11, 97.46) mm, rotated rx -180 ry 0 rz 180 deg; joints [-169.147, 62.59, -80.877, 168.584, 72.051, 3.561]
  Call Extruder(75.65986)
  MoveL 6497 to (-22.56, 35.07, 97.46) mm, rotated rx -180 ry 0 rz -180 deg; joints [-169.127, 62.543, -80.902, 168.559, 71.982, 3.582]
  MoveL 6498 to (-22.56, 35.07, 97.46) mm, rotated rx -180 ry 0 rz -180 deg; joints [-169.127, 62.543, -80.902, 168.559, 71.982, 3.582]
  Call Extruder(75.95325)
  MoveL 6499 to (-21.97, 35.02, 97.46) mm, rotated rx 180 ry 0 rz 180 deg; joints [-169.107, 62.495, -80.926, 168.533, 71.912, 3.604]
  MoveL 6500 to (-21.97, 35.02, 97.46) mm, rotated rx 180 ry 0 rz 180 deg; joints [-169.107, 62.495, -80.926, 168.533, 71.912, 3.604]
  Call Extruder(76.38658)
  MoveL 6501 to (-21.1, 34.97, 97.46) mm, rotated rx -180 ry 0 rz -180 deg; joints [-169.069, 62.425, -80.963, 168.487, 71.81, 3.638]
  MoveL 6502 to (-21.1, 34.97, 97.46) mm, rotated rx -180 ry 0 rz -180 deg; joints [-169.069, 62.425, -80.963, 168.487, 71.81, 3.638]
  Call Extruder(76.95874)
  MoveL 6503 to (-19.94, 34.93, 97.46) mm, rotated rx -180 ry 0 rz -180 deg; joints [-169.014, 62.331, -81.01, 168.419, 71.676, 3.686]
  MoveL 6504 to (-19.94, 34.93, 97.46) mm, rotated rx -180 ry 0 rz -180 deg; joints [-169.014, 62.331, -81.01, 168.419, 71.676, 3.686]
  Call Extruder(77.38658)
  MoveL 6505 to (-19.06, 34.91, 97.46) mm, rotated rx 180 ry 0 rz 180 deg; joints [-168.967, 62.261, -81.045, 168.363, 71.575, 3.724]
  Call Extruder(194.03526)
  MoveL 6506 to (219.06, 34.91, 97.46) mm, rotated rx -180 ry 0 rz 180 deg; joints [-30.588, 51.226, -83.228, 34.878, 117.143, 17.641]
  MoveL 6507 to (219.06, 34.91, 97.46) mm, rotated rx -180 ry 0 rz 180 deg; joints [-30.588, 51.226, -83.228, 34.878, 117.143, 17.641]
  Call Extruder(194.75084)
  MoveL 6508 to (220.52, 34.95, 97.46) mm, rotated rx -180 ry 0 rz 180 deg; joints [-30.009, 51.367, -83.231, 34.217, 117.203, 17.269]
  MoveL 6509 to (220.52, 34.95, 97.46) mm, rotated rx -180 ry 0 rz 180 deg; joints [-30.009, 51.367, -83.231, 34.217, 117.203, 17.269]
  Call Extruder(195.32557)
  MoveL 6510 to (221.68, 35, 97.46) mm, rotated rx 180 ry 0 rz 180 deg; joints [-29.572, 51.481, -83.233, 33.715, 117.239, 16.984]
  MoveL 6511 to (221.68, 35, 97.46) mm, rotated rx 180 ry 0 rz 180 deg; joints [-29.572, 51.481, -83.233, 33.715, 117.239, 16.984]
  Call Extruder(195.61897)
  MoveL 6512 to (222.27, 35.05, 97.46) mm, rotated rx 180 ry 0 rz 180 deg; joints [-29.371, 51.54, -83.234, 33.482, 117.248, 16.848]
  MoveL 6513 to (222.27, 35.05, 97.46) mm, rotated rx 180 ry 0 rz 180 deg; joints [-29.371, 51.54, -83.234, 33.482, 117.248, 16.848]
  Call Extruder(195.91369)
  MoveL 6514 to (222.86, 35.09, 97.46) mm, rotated rx 180 ry 0 rz -180 deg; joints [-29.173, 51.599, -83.234, 33.253, 117.257, 16.715]
  MoveL 6515 to (222.86, 35.09, 97.46) mm, rotated rx 180 ry 0 rz -180 deg; joints [-29.173, 51.599, -83.234, 33.253, 117.257, 16.715]
  Call Extruder(196.20975)
  MoveL 6516 to (223.45, 35.14, 97.46) mm, rotated rx -180 ry 0 rz 180 deg; joints [-28.978, 51.658, -83.235, 33.026, 117.264, 16.583]
  MoveL 6517 to (223.45, 35.14, 97.46) mm, rotated rx -180 ry 0 rz 180 deg; joints [-28.978, 51.658, -83.235, 33.026, 117.264, 16.583]
  Call Extruder(196.40603)
  MoveL 6518 to (223.84, 35.18, 97.46) mm, rotated rx 180 ry 0 rz 180 deg; joints [-28.862, 51.698, -83.235, 32.89, 117.264, 16.501]
  MoveL 6519 to (223.84, 35.18, 97.46) mm, rotated rx 180 ry 0 rz 180 deg; joints [-28.862, 51.698, -83.235, 32.89, 117.264, 16.501]
  Call Extruder(196.60317)
  MoveL 6520 to (224.22, 35.23, 97.46) mm, rotated rx -180 ry 0 rz 180 deg; joints [-28.747, 51.737, -83.236, 32.754, 117.263, 16.42]
  MoveL 6521 to (224.22, 35.23, 97.46) mm, rotated rx -180 ry 0 rz 180 deg; joints [-28.747, 51.737, -83.236, 32.754, 117.263, 16.42]
  Call Extruder(196.80118)
  MoveL 6522 to (224.61, 35.27, 97.46) mm, rotated rx -180 ry 0 rz 180 deg; joints [-28.633, 51.777, -83.236, 32.621, 117.262, 16.34]
  MoveL 6523 to (224.61, 35.27, 97.46) mm, rotated rx -180 ry 0 rz 180 deg; joints [-28.633, 51.777, -83.236, 32.621, 117.262, 16.34]
  Call Extruder(197.00005)
  MoveL 6524 to (225, 35.32, 97.46) mm, rotated rx 180 ry 0 rz 180 deg; joints [-28.52, 51.817, -83.236, 32.488, 117.26, 16.26]
  MoveL 6525 to (225, 35.32, 97.46) mm, rotated rx 180 ry 0 rz 180 deg; joints [-28.52, 51.817, -83.236, 32.488, 117.26, 16.26]
  Call Extruder(197.17913)
  MoveL 6526 to (225.34, 35.37, 97.46) mm, rotated rx -180 ry 0 rz -180 deg; joints [-28.425, 51.852, -83.236, 32.375, 117.257, 16.192]
  MoveL 6527 to (225.34, 35.37, 97.46) mm, rotated rx -180 ry 0 rz -180 deg; joints [-28.425, 51.852, -83.236, 32.375, 117.257, 16.192]
  Call Extruder(197.33832)
  MoveL 6528 to (225.65, 35.42, 97.46) mm, rotated rx 180 ry 0 rz 180 deg; joints [-28.346, 51.884, -83.236, 32.281, 117.252, 16.133]
  MoveL 6529 to (225.65, 35.42, 97.46) mm, rotated rx 180 ry 0 rz 180 deg; joints [-28.346, 51.884, -83.236, 32.281, 117.252, 16.133]
  Call Extruder(197.49823)
  MoveL 6530 to (225.96, 35.47, 97.46) mm, rotated rx -180 ry 0 rz -180 deg; joints [-28.267, 51.916, -83.236, 32.187, 117.247, 16.075]
  MoveL 6531 to (225.96, 35.47, 97.46) mm, rotated rx -180 ry 0 rz -180 deg; joints [-28.267, 51.916, -83.236, 32.187, 117.247, 16.075]
  Call Extruder(197.65887)
  MoveL 6532 to (226.26, 35.51, 97.46) mm, rotated rx 180 ry 0 rz 180 deg; joints [-28.19, 51.948, -83.236, 32.095, 117.241, 16.018]
  MoveL 6533 to (226.26, 35.51, 97.46) mm, rotated rx 180 ry 0 rz 180 deg; joints [-28.19, 51.948, -83.236, 32.095, 117.241, 16.018]
  Call Extruder(197.82023)
  MoveL 6534 to (226.57, 35.56, 97.46) mm, rotated rx 180 ry 0 rz -180 deg; joints [-28.112, 51.98, -83.236, 32.003, 117.235, 15.96]
  MoveL 6535 to (226.57, 35.56, 97.46) mm, rotated rx 180 ry 0 rz -180 deg; joints [-28.112, 51.98, -83.236, 32.003, 117.235, 15.96]
  Call Extruder(197.98233)
  MoveL 6536 to (226.87, 35.61, 97.46) mm, rotated rx 180 ry 0 rz 180 deg; joints [-28.036, 52.012, -83.236, 31.911, 117.229, 15.904]
  MoveL 6537 to (226.87, 35.61, 97.46) mm, rotated rx 180 ry 0 rz 180 deg; joints [-28.036, 52.012, -83.236, 31.911, 117.229, 15.904]
  Call Extruder(198.13052)
  MoveL 6538 to (227.15, 35.66, 97.46) mm, rotated rx -180 ry 0 rz 180 deg; joints [-27.971, 52.041, -83.236, 31.832, 117.222, 15.854]
  MoveL 6539 to (227.15, 35.66, 97.46) mm, rotated rx -180 ry 0 rz 180 deg; joints [-27.971, 52.041, -83.236, 31.832, 117.222, 15.854]
  Call Extruder(198.26476)
  MoveL 6540 to (227.4, 35.71, 97.46) mm, rotated rx -180 ry 0 rz 180 deg; joints [-27.915, 52.068, -83.236, 31.765, 117.215, 15.811]
  MoveL 6541 to (227.4, 35.71, 97.46) mm, rotated rx -180 ry 0 rz 180 deg; joints [-27.915, 52.068, -83.236, 31.765, 117.215, 15.811]
  Call Extruder(198.39960)
  MoveL 6542 to (227.65, 35.76, 97.46) mm, rotated rx 180 ry 0 rz 180 deg; joints [-27.861, 52.094, -83.236, 31.7, 117.207, 15.768]
  MoveL 6543 to (227.65, 35.76, 97.46) mm, rotated rx 180 ry 0 rz 180 deg; joints [-27.861, 52.094, -83.236, 31.7, 117.207, 15.768]
  Call Extruder(198.53505)
  MoveL 6544 to (227.9, 35.81, 97.46) mm, rotated rx -180 ry 0 rz -180 deg; joints [-27.807, 52.121, -83.236, 31.633, 117.199, 15.725]
  MoveL 6545 to (227.9, 35.81, 97.46) mm, rotated rx -180 ry 0 rz -180 deg; joints [-27.807, 52.121, -83.236, 31.633, 117.199, 15.725]
  Call Extruder(198.67111)
  MoveL 6546 to (228.15, 35.86, 97.46) mm, rotated rx 180 ry 0 rz 180 deg; joints [-27.753, 52.147, -83.235, 31.568, 117.191, 15.683]
  MoveL 6547 to (228.15, 35.86, 97.46) mm, rotated rx 180 ry 0 rz 180 deg; joints [-27.753, 52.147, -83.235, 31.568, 117.191, 15.683]
  Call Extruder(198.80779)
  MoveL 6548 to (228.4, 35.91, 97.46) mm, rotated rx -180 ry 0 rz 180 deg; joints [-27.699, 52.174, -83.235, 31.502, 117.183, 15.641]
  MoveL 6549 to (228.4, 35.91, 97.46) mm, rotated rx -180 ry 0 rz 180 deg; joints [-27.699, 52.174, -83.235, 31.502, 117.183, 15.641]
  Call Extruder(198.94507)
  MoveL 6550 to (228.65, 35.96, 97.46) mm, rotated rx -180 ry 0 rz -180 deg; joints [-27.646, 52.2, -83.235, 31.438, 117.174, 15.599]
  MoveL 6551 to (228.65, 35.96, 97.46) mm, rotated rx -180 ry 0 rz -180 deg; joints [-27.646, 52.2, -83.235, 31.438, 117.174, 15.599]
  Call Extruder(199.07074)
  MoveL 6552 to (228.87, 36, 97.46) mm, rotated rx -180 ry 0 rz 180 deg; joints [-27.599, 52.225, -83.235, 31.381, 117.166, 15.562]
  MoveL 6553 to (228.87, 36, 97.46) mm, rotated rx -180 ry 0 rz 180 deg; joints [-27.599, 52.225, -83.235, 31.381, 117.166, 15.562]
  Call Extruder(199.18469)
  MoveL 6554 to (229.08, 36.05, 97.46) mm, rotated rx -180 ry 0 rz 180 deg; joints [-27.559, 52.247, -83.235, 31.331, 117.158, 15.529]
  MoveL 6555 to (229.08, 36.05, 97.46) mm, rotated rx -180 ry 0 rz 180 deg; joints [-27.559, 52.247, -83.235, 31.331, 117.158, 15.529]
  Call Extruder(199.29908)
  MoveL 6556 to (229.28, 36.09, 97.46) mm, rotated rx 180 ry 0 rz 180 deg; joints [-27.518, 52.268, -83.234, 31.281, 117.15, 15.496]
  MoveL 6557 to (229.28, 36.09, 97.46) mm, rotated rx 180 ry 0 rz 180 deg; joints [-27.518, 52.268, -83.234, 31.281, 117.15, 15.496]
  Call Extruder(199.41393)
  MoveL 6558 to (229.48, 36.14, 97.46) mm, rotated rx 180 ry 0 rz 180 deg; joints [-27.479, 52.29, -83.234, 31.233, 117.141, 15.463]
  MoveL 6559 to (229.48, 36.14, 97.46) mm, rotated rx 180 ry 0 rz 180 deg; joints [-27.479, 52.29, -83.234, 31.233, 117.141, 15.463]
  Call Extruder(199.52924)
  MoveL 6560 to (229.69, 36.18, 97.46) mm, rotated rx 180 ry 0 rz 180 deg; joints [-27.439, 52.312, -83.234, 31.184, 117.133, 15.431]
  MoveL 6561 to (229.69, 36.18, 97.46) mm, rotated rx 180 ry 0 rz 180 deg; joints [-27.439, 52.312, -83.234, 31.184, 117.133, 15.431]
  Call Extruder(199.65360)
  MoveL 6562 to (229.9, 36.25, 97.46) mm, rotated rx 180 ry 0 rz 180 deg; joints [-27.408, 52.336, -83.233, 31.144, 117.12, 15.401]
  MoveL 6563 to (229.9, 36.25, 97.46) mm, rotated rx 180 ry 0 rz 180 deg; joints [-27.408, 52.336, -83.233, 31.144, 117.12, 15.401]
  Call Extruder(199.77848)
  MoveL 6564 to (230.12, 36.31, 97.46) mm, rotated rx -180 ry 0 rz 180 deg; joints [-27.377, 52.36, -83.233, 31.104, 117.108, 15.372]
  MoveL 6565 to (230.12, 36.31, 97.46) mm, rotated rx -180 ry 0 rz 180 deg; joints [-27.377, 52.36, -83.233, 31.104, 117.108, 15.372]
  Call Extruder(199.90388)
  MoveL 6566 to (230.33, 36.38, 97.46) mm, rotated rx -180 ry 0 rz 180 deg; joints [-27.348, 52.384, -83.233, 31.065, 117.095, 15.343]
  MoveL 6567 to (230.33, 36.38, 97.46) mm, rotated rx -180 ry 0 rz 180 deg; joints [-27.348, 52.384, -83.233, 31.065, 117.095, 15.343]
  Call Extruder(200.02979)
  MoveL 6568 to (230.55, 36.44, 97.46) mm, rotated rx -180 ry 0 rz -180 deg; joints [-27.317, 52.408, -83.232, 31.026, 117.082, 15.314]
  MoveL 6569 to (230.55, 36.44, 97.46) mm, rotated rx -180 ry 0 rz -180 deg; joints [-27.317, 52.408, -83.232, 31.026, 117.082, 15.314]
  Call Extruder(200.11575)
  MoveL 6570 to (230.7, 36.49, 97.46) mm, rotated rx -180 ry 0 rz 180 deg; joints [-27.299, 52.424, -83.232, 31.002, 117.073, 15.296]
  MoveL 6571 to (230.7, 36.49, 97.46) mm, rotated rx -180 ry 0 rz 180 deg; joints [-27.299, 52.424, -83.232, 31.002, 117.073, 15.296]
  Call Extruder(200.22765)
  MoveL 6572 to (230.88, 36.55, 97.46) mm, rotated rx 180 ry 0 rz 180 deg; joints [-27.276, 52.445, -83.232, 30.972, 117.06, 15.272]
  MoveL 6573 to (230.88, 36.55, 97.46) mm, rotated rx 180 ry 0 rz 180 deg; joints [-27.276, 52.445, -83.232, 30.972, 117.06, 15.272]
  Call Extruder(200.33999)
  MoveL 6574 to (231.07, 36.61, 97.46) mm, rotated rx -180 ry 0 rz 180 deg; joints [-27.253, 52.467, -83.231, 30.941, 117.048, 15.248]
  MoveL 6575 to (231.07, 36.61, 97.46) mm, rotated rx -180 ry 0 rz 180 deg; joints [-27.253, 52.467, -83.231, 30.941, 117.048, 15.248]
  Call Extruder(200.45278)
  MoveL 6576 to (231.26, 36.67, 97.46) mm, rotated rx -180 ry 0 rz 180 deg; joints [-27.231, 52.488, -83.231, 30.911, 117.035, 15.225]
  MoveL 6577 to (231.26, 36.67, 97.46) mm, rotated rx -180 ry 0 rz 180 deg; joints [-27.231, 52.488, -83.231, 30.911, 117.035, 15.225]
  Call Extruder(200.56601)
  MoveL 6578 to (231.45, 36.73, 97.46) mm, rotated rx -180 ry 0 rz 180 deg; joints [-27.208, 52.509, -83.231, 30.881, 117.023, 15.201]
  MoveL 6579 to (231.45, 36.73, 97.46) mm, rotated rx -180 ry 0 rz 180 deg; joints [-27.208, 52.509, -83.231, 30.881, 117.023, 15.201]
  Call Extruder(200.67969)
  MoveL 6580 to (231.64, 36.79, 97.46) mm, rotated rx -180 ry 0 rz 180 deg; joints [-27.185, 52.53, -83.23, 30.851, 117.01, 15.177]
  MoveL 6581 to (231.64, 36.79, 97.46) mm, rotated rx -180 ry 0 rz 180 deg; joints [-27.185, 52.53, -83.23, 30.851, 117.01, 15.177]
  Call Extruder(200.86165)
  MoveL 6582 to (231.93, 36.91, 97.46) mm, rotated rx 180 ry 0 rz -180 deg; joints [-27.167, 52.564, -83.23, 30.822, 116.985, 15.148]
  MoveL 6583 to (231.93, 36.91, 97.46) mm, rotated rx 180 ry 0 rz -180 deg; joints [-27.167, 52.564, -83.23, 30.822, 116.985, 15.148]
  Call Extruder(201.04437)
  MoveL 6584 to (232.22, 37.04, 97.46) mm, rotated rx 180 ry 0 rz -180 deg; joints [-27.149, 52.598, -83.229, 30.793, 116.96, 15.12]
  MoveL 6585 to (232.22, 37.04, 97.46) mm, rotated rx 180 ry 0 rz -180 deg; joints [-27.149, 52.598, -83.229, 30.793, 116.96, 15.12]
  Call Extruder(201.21479)
  MoveL 6586 to (232.49, 37.15, 97.46) mm, rotated rx -180 ry 0 rz 180 deg; joints [-27.133, 52.63, -83.228, 30.768, 116.936, 15.094]
  MoveL 6587 to (232.49, 37.15, 97.46) mm, rotated rx -180 ry 0 rz 180 deg; joints [-27.133, 52.63, -83.228, 30.768, 116.936, 15.094]
  Call Extruder(201.37278)
  MoveL 6588 to (232.74, 37.26, 97.46) mm, rotated rx 180 ry 0 rz 180 deg; joints [-27.121, 52.659, -83.228, 30.746, 116.914, 15.07]
  MoveL 6589 to (232.74, 37.26, 97.46) mm, rotated rx 180 ry 0 rz 180 deg; joints [-27.121, 52.659, -83.228, 30.746, 116.914, 15.07]
  Call Extruder(201.53139)
  MoveL 6590 to (232.99, 37.36, 97.46) mm, rotated rx -180 ry 0 rz 180 deg; joints [-27.108, 52.688, -83.227, 30.724, 116.892, 15.047]
  MoveL 6591 to (232.99, 37.36, 97.46) mm, rotated rx -180 ry 0 rz 180 deg; joints [-27.108, 52.688, -83.227, 30.724, 116.892, 15.047]
  Call Extruder(201.73755)
  MoveL 6592 to (233.29, 37.54, 97.46) mm, rotated rx 180 ry 0 rz 180 deg; joints [-27.12, 52.726, -83.226, 30.727, 116.855, 15.03]
  MoveL 6593 to (233.29, 37.54, 97.46) mm, rotated rx 180 ry 0 rz 180 deg; joints [-27.12, 52.726, -83.226, 30.727, 116.855, 15.03]
  Call Extruder(201.94450)
  MoveL 6594 to (233.6, 37.71, 97.46) mm, rotated rx -180 ry 0 rz 180 deg; joints [-27.132, 52.764, -83.225, 30.731, 116.819, 15.014]
  MoveL 6595 to (233.6, 37.71, 97.46) mm, rotated rx -180 ry 0 rz 180 deg; joints [-27.132, 52.764, -83.225, 30.731, 116.819, 15.014]
  Call Extruder(202.15222)
  MoveL 6596 to (233.9, 37.89, 97.46) mm, rotated rx -180 ry 0 rz 180 deg; joints [-27.144, 52.801, -83.224, 30.734, 116.782, 14.998]
  MoveL 6597 to (233.9, 37.89, 97.46) mm, rotated rx -180 ry 0 rz 180 deg; joints [-27.144, 52.801, -83.224, 30.734, 116.782, 14.998]
  Call Extruder(202.36072)
  MoveL 6598 to (234.21, 38.06, 97.46) mm, rotated rx -180 ry 0 rz 180 deg; joints [-27.156, 52.839, -83.223, 30.737, 116.746, 14.982]
  MoveL 6599 to (234.21, 38.06, 97.46) mm, rotated rx -180 ry 0 rz 180 deg; joints [-27.156, 52.839, -83.223, 30.737, 116.746, 14.982]
  Call Extruder(202.54027)
  MoveL 6600 to (234.45, 38.24, 97.46) mm, rotated rx -180 ry 0 rz 180 deg; joints [-27.187, 52.871, -83.222, 30.762, 116.71, 14.978]
  MoveL 6601 to (234.45, 38.24, 97.46) mm, rotated rx -180 ry 0 rz 180 deg; joints [-27.187, 52.871, -83.222, 30.762, 116.71, 14.978]
  Call Extruder(202.87368)
  MoveL 6602 to (234.9, 38.57, 97.46) mm, rotated rx -180 ry 0 rz 180 deg; joints [-27.245, 52.93, -83.22, 30.809, 116.642, 14.971]
  MoveL 6603 to (234.9, 38.57, 97.46) mm, rotated rx -180 ry 0 rz 180 deg; joints [-27.245, 52.93, -83.22, 30.809, 116.642, 14.971]
  Call Extruder(203.20828)
  MoveL 6604 to (235.35, 38.9, 97.46) mm, rotated rx -180 ry 0 rz 180 deg; joints [-27.302, 52.989, -83.218, 30.855, 116.575, 14.964]
  Call Extruder(204.03623)
  MoveL 6605 to (236.39, 39.81, 97.46) mm, rotated rx -180 ry 0 rz 180 deg; joints [-27.525, 53.133, -83.213, 31.057, 116.39, 14.985]
  Call Extruder(204.86417)
  MoveL 6606 to (237.3, 40.85, 97.46) mm, rotated rx 180 ry 0 rz 180 deg; joints [-27.851, 53.27, -83.207, 31.372, 116.183, 15.058]
  Call Extruder(205.03147)
  MoveL 6607 to (237.47, 41.07, 97.46) mm, rotated rx -180 ry 0 rz 180 deg; joints [-27.932, 53.297, -83.206, 31.452, 116.138, 15.08]
  MoveL 6608 to (237.47, 41.07, 97.46) mm, rotated rx -180 ry 0 rz 180 deg; joints [-27.932, 53.297, -83.206, 31.452, 116.138, 15.08]
  Call Extruder(205.36489)
  MoveL 6609 to (237.8, 41.52, 97.46) mm, rotated rx -180 ry 0 rz 180 deg; joints [-28.091, 53.35, -83.203, 31.609, 116.049, 15.123]
  MoveL 6610 to (237.8, 41.52, 97.46) mm, rotated rx -180 ry 0 rz 180 deg; joints [-28.091, 53.35, -83.203, 31.609, 116.049, 15.123]
  Call Extruder(205.69712)
  MoveL 6611 to (238.12, 41.98, 97.46) mm, rotated rx 180 ry 0 rz -180 deg; joints [-28.249, 53.404, -83.201, 31.763, 115.96, 15.164]
  MoveL 6612 to (238.12, 41.98, 97.46) mm, rotated rx 180 ry 0 rz -180 deg; joints [-28.249, 53.404, -83.201, 31.763, 115.96, 15.164]
  Call Extruder(205.81481)
  MoveL 6613 to (238.22, 42.15, 97.46) mm, rotated rx -180 ry 0 rz -180 deg; joints [-28.315, 53.422, -83.2, 31.83, 115.927, 15.185]
  MoveL 6614 to (238.22, 42.15, 97.46) mm, rotated rx -180 ry 0 rz -180 deg; joints [-28.315, 53.422, -83.2, 31.83, 115.927, 15.185]
  Call Extruder(206.02254)
  MoveL 6615 to (238.4, 42.45, 97.46) mm, rotated rx -180 ry 0 rz 180 deg; joints [-28.434, 53.453, -83.198, 31.949, 115.867, 15.221]
  MoveL 6616 to (238.4, 42.45, 97.46) mm, rotated rx -180 ry 0 rz 180 deg; joints [-28.434, 53.453, -83.198, 31.949, 115.867, 15.221]
  Call Extruder(206.22948)
  MoveL 6617 to (238.57, 42.75, 97.46) mm, rotated rx -180 ry 0 rz 180 deg; joints [-28.552, 53.485, -83.196, 32.067, 115.808, 15.256]
  MoveL 6618 to (238.57, 42.75, 97.46) mm, rotated rx -180 ry 0 rz 180 deg; joints [-28.552, 53.485, -83.196, 32.067, 115.808, 15.256]
  Call Extruder(206.43565)
  MoveL 6619 to (238.75, 43.06, 97.46) mm, rotated rx 180 ry 0 rz 180 deg; joints [-28.669, 53.517, -83.195, 32.183, 115.749, 15.291]
  MoveL 6620 to (238.75, 43.06, 97.46) mm, rotated rx 180 ry 0 rz 180 deg; joints [-28.669, 53.517, -83.195, 32.183, 115.749, 15.291]
  Call Extruder(206.61734)
  MoveL 6621 to (238.89, 43.34, 97.46) mm, rotated rx 180 ry 0 rz 180 deg; joints [-28.78, 53.544, -83.193, 32.295, 115.695, 15.326]
  MoveL 6622 to (238.89, 43.34, 97.46) mm, rotated rx 180 ry 0 rz 180 deg; joints [-28.78, 53.544, -83.193, 32.295, 115.695, 15.326]
  Call Extruder(206.77535)
  MoveL 6623 to (239, 43.58, 97.46) mm, rotated rx -180 ry 0 rz 180 deg; joints [-28.886, 53.567, -83.192, 32.402, 115.647, 15.36]
  MoveL 6624 to (239, 43.58, 97.46) mm, rotated rx -180 ry 0 rz 180 deg; joints [-28.886, 53.567, -83.192, 32.402, 115.647, 15.36]
  Call Extruder(206.93276)
  MoveL 6625 to (239.11, 43.83, 97.46) mm, rotated rx -180 ry 0 rz -180 deg; joints [-28.991, 53.589, -83.191, 32.509, 115.599, 15.395]
  MoveL 6626 to (239.11, 43.83, 97.46) mm, rotated rx -180 ry 0 rz -180 deg; joints [-28.991, 53.589, -83.191, 32.509, 115.599, 15.395]
  Call Extruder(207.11547)
  MoveL 6627 to (239.23, 44.13, 97.46) mm, rotated rx 180 ry 0 rz 180 deg; joints [-29.116, 53.615, -83.189, 32.635, 115.542, 15.436]
  MoveL 6628 to (239.23, 44.13, 97.46) mm, rotated rx 180 ry 0 rz 180 deg; joints [-29.116, 53.615, -83.189, 32.635, 115.542, 15.436]
  Call Extruder(207.29743)
  MoveL 6629 to (239.35, 44.42, 97.46) mm, rotated rx -180 ry 0 rz 180 deg; joints [-29.24, 53.642, -83.188, 32.76, 115.486, 15.476]
  MoveL 6630 to (239.35, 44.42, 97.46) mm, rotated rx -180 ry 0 rz 180 deg; joints [-29.24, 53.642, -83.188, 32.76, 115.486, 15.476]
  Call Extruder(207.44476)
  MoveL 6631 to (239.44, 44.66, 97.46) mm, rotated rx -180 ry 0 rz 180 deg; joints [-29.343, 53.663, -83.187, 32.865, 115.44, 15.511]
  MoveL 6632 to (239.44, 44.66, 97.46) mm, rotated rx -180 ry 0 rz 180 deg; joints [-29.343, 53.663, -83.187, 32.865, 115.44, 15.511]
  Call Extruder(207.55800)
  MoveL 6633 to (239.5, 44.85, 97.46) mm, rotated rx 180 ry 0 rz 180 deg; joints [-29.428, 53.678, -83.186, 32.951, 115.404, 15.539]
  MoveL 6634 to (239.5, 44.85, 97.46) mm, rotated rx 180 ry 0 rz 180 deg; joints [-29.428, 53.678, -83.186, 32.951, 115.404, 15.539]
  Call Extruder(207.67079)
  MoveL 6635 to (239.56, 45.03, 97.46) mm, rotated rx -180 ry 0 rz 180 deg; joints [-29.512, 53.693, -83.185, 33.036, 115.367, 15.568]
  MoveL 6636 to (239.56, 45.03, 97.46) mm, rotated rx -180 ry 0 rz 180 deg; joints [-29.512, 53.693, -83.185, 33.036, 115.367, 15.568]
  Call Extruder(207.78314)
  MoveL 6637 to (239.62, 45.22, 97.46) mm, rotated rx 180 ry 0 rz -180 deg; joints [-29.596, 53.709, -83.184, 33.121, 115.331, 15.596]
  MoveL 6638 to (239.62, 45.22, 97.46) mm, rotated rx 180 ry 0 rz -180 deg; joints [-29.596, 53.709, -83.184, 33.121, 115.331, 15.596]
  Call Extruder(207.89504)
  MoveL 6639 to (239.68, 45.41, 97.46) mm, rotated rx 180 ry 0 rz 180 deg; joints [-29.679, 53.724, -83.183, 33.206, 115.295, 15.625]
  MoveL 6640 to (239.68, 45.41, 97.46) mm, rotated rx 180 ry 0 rz 180 deg; joints [-29.679, 53.724, -83.183, 33.206, 115.295, 15.625]
  Call Extruder(208.01644)
  MoveL 6641 to (239.75, 45.62, 97.46) mm, rotated rx -180 ry 0 rz 180 deg; joints [-29.77, 53.741, -83.182, 33.299, 115.256, 15.655]
  MoveL 6642 to (239.75, 45.62, 97.46) mm, rotated rx -180 ry 0 rz 180 deg; joints [-29.77, 53.741, -83.182, 33.299, 115.256, 15.655]
  Call Extruder(208.14723)
  MoveL 6643 to (239.82, 45.84, 97.46) mm, rotated rx 180 ry 0 rz 180 deg; joints [-29.871, 53.759, -83.181, 33.4, 115.213, 15.689]
  MoveL 6644 to (239.82, 45.84, 97.46) mm, rotated rx 180 ry 0 rz 180 deg; joints [-29.871, 53.759, -83.181, 33.4, 115.213, 15.689]
  Call Extruder(208.27745)
  MoveL 6645 to (239.88, 46.06, 97.46) mm, rotated rx 180 ry 0 rz -180 deg; joints [-29.97, 53.777, -83.18, 33.501, 115.17, 15.723]
  MoveL 6646 to (239.88, 46.06, 97.46) mm, rotated rx 180 ry 0 rz -180 deg; joints [-29.97, 53.777, -83.18, 33.501, 115.17, 15.723]
  Call Extruder(208.40711)
  MoveL 6647 to (239.95, 46.29, 97.46) mm, rotated rx -180 ry 0 rz 180 deg; joints [-30.069, 53.795, -83.179, 33.602, 115.127, 15.756]
  MoveL 6648 to (239.95, 46.29, 97.46) mm, rotated rx -180 ry 0 rz 180 deg; joints [-30.069, 53.795, -83.179, 33.602, 115.127, 15.756]
  Call Extruder(208.53621)
  MoveL 6649 to (240.02, 46.51, 97.46) mm, rotated rx 180 ry 0 rz -180 deg; joints [-30.168, 53.813, -83.178, 33.702, 115.084, 15.789]
  MoveL 6650 to (240.02, 46.51, 97.46) mm, rotated rx 180 ry 0 rz -180 deg; joints [-30.168, 53.813, -83.178, 33.702, 115.084, 15.789]
  Call Extruder(208.65126)
  MoveL 6651 to (240.06, 46.72, 97.46) mm, rotated rx -180 ry 0 rz 180 deg; joints [-30.263, 53.828, -83.177, 33.799, 115.045, 15.822]
  MoveL 6652 to (240.06, 46.72, 97.46) mm, rotated rx -180 ry 0 rz 180 deg; joints [-30.263, 53.828, -83.177, 33.799, 115.045, 15.822]
  Call Extruder(208.76586)
  MoveL 6653 to (240.11, 46.92, 97.46) mm, rotated rx -180 ry 0 rz -180 deg; joints [-30.358, 53.843, -83.176, 33.895, 115.006, 15.855]
  MoveL 6654 to (240.11, 46.92, 97.46) mm, rotated rx -180 ry 0 rz -180 deg; joints [-30.358, 53.843, -83.176, 33.895, 115.006, 15.855]
  Call Extruder(208.88001)
  MoveL 6655 to (240.15, 47.12, 97.46) mm, rotated rx -180 ry 0 rz 180 deg; joints [-30.453, 53.857, -83.175, 33.992, 114.967, 15.887]
  MoveL 6656 to (240.15, 47.12, 97.46) mm, rotated rx -180 ry 0 rz 180 deg; joints [-30.453, 53.857, -83.175, 33.992, 114.967, 15.887]
  Call Extruder(208.99371)
  MoveL 6657 to (240.2, 47.33, 97.46) mm, rotated rx -180 ry 0 rz 180 deg; joints [-30.548, 53.873, -83.174, 34.088, 114.928, 15.92]
  MoveL 6658 to (240.2, 47.33, 97.46) mm, rotated rx -180 ry 0 rz 180 deg; joints [-30.548, 53.873, -83.174, 34.088, 114.928, 15.92]
  Call Extruder(209.11912)
  MoveL 6659 to (240.24, 47.55, 97.46) mm, rotated rx -180 ry 0 rz 180 deg; joints [-30.653, 53.889, -83.173, 34.195, 114.885, 15.956]
  MoveL 6660 to (240.24, 47.55, 97.46) mm, rotated rx -180 ry 0 rz 180 deg; joints [-30.653, 53.889, -83.173, 34.195, 114.885, 15.956]
  Call Extruder(209.25610)
  MoveL 6661 to (240.29, 47.8, 97.46) mm, rotated rx -180 ry 0 rz 180 deg; joints [-30.768, 53.907, -83.171, 34.312, 114.837, 15.996]
  MoveL 6662 to (240.29, 47.8, 97.46) mm, rotated rx -180 ry 0 rz 180 deg; joints [-30.768, 53.907, -83.171, 34.312, 114.837, 15.996]
  Call Extruder(209.39246)
  MoveL 6663 to (240.34, 48.05, 97.46) mm, rotated rx 180 ry 0 rz 180 deg; joints [-30.884, 53.925, -83.17, 34.43, 114.789, 16.035]
  MoveL 6664 to (240.34, 48.05, 97.46) mm, rotated rx 180 ry 0 rz 180 deg; joints [-30.884, 53.925, -83.17, 34.43, 114.789, 16.035]
  Call Extruder(209.52822)
  MoveL 6665 to (240.39, 48.3, 97.46) mm, rotated rx 180 ry 0 rz -180 deg; joints [-30.999, 53.943, -83.169, 34.547, 114.742, 16.074]
  MoveL 6666 to (240.39, 48.3, 97.46) mm, rotated rx 180 ry 0 rz -180 deg; joints [-30.999, 53.943, -83.169, 34.547, 114.742, 16.074]
  Call Extruder(209.66337)
  MoveL 6667 to (240.44, 48.55, 97.46) mm, rotated rx -180 ry 0 rz 180 deg; joints [-31.114, 53.961, -83.168, 34.663, 114.694, 16.113]
  MoveL 6668 to (240.44, 48.55, 97.46) mm, rotated rx -180 ry 0 rz 180 deg; joints [-31.114, 53.961, -83.168, 34.663, 114.694, 16.113]
  Call Extruder(209.79791)
  MoveL 6669 to (240.49, 48.8, 97.46) mm, rotated rx -180 ry 0 rz 180 deg; joints [-31.228, 53.979, -83.167, 34.779, 114.646, 16.151]
  MoveL 6670 to (240.49, 48.8, 97.46) mm, rotated rx -180 ry 0 rz 180 deg; joints [-31.228, 53.979, -83.167, 34.779, 114.646, 16.151]
  Call Extruder(209.93183)
  MoveL 6671 to (240.54, 49.05, 97.46) mm, rotated rx -180 ry 0 rz 180 deg; joints [-31.342, 53.997, -83.165, 34.894, 114.599, 16.189]
  MoveL 6672 to (240.54, 49.05, 97.46) mm, rotated rx -180 ry 0 rz 180 deg; joints [-31.342, 53.997, -83.165, 34.894, 114.599, 16.189]
  Call Extruder(210.07970)
  MoveL 6673 to (240.59, 49.33, 97.46) mm, rotated rx 180 ry 0 rz 180 deg; joints [-31.47, 54.016, -83.164, 35.024, 114.546, 16.233]
  MoveL 6674 to (240.59, 49.33, 97.46) mm, rotated rx 180 ry 0 rz 180 deg; joints [-31.47, 54.016, -83.164, 35.024, 114.546, 16.233]
  Call Extruder(210.24144)
  MoveL 6675 to (240.64, 49.63, 97.46) mm, rotated rx -180 ry 0 rz 180 deg; joints [-31.612, 54.037, -83.162, 35.168, 114.488, 16.281]
  MoveL 6676 to (240.64, 49.63, 97.46) mm, rotated rx -180 ry 0 rz 180 deg; joints [-31.612, 54.037, -83.162, 35.168, 114.488, 16.281]
  Call Extruder(210.40246)
  MoveL 6677 to (240.69, 49.94, 97.46) mm, rotated rx -180 ry 0 rz 180 deg; joints [-31.755, 54.058, -83.161, 35.312, 114.429, 16.328]
  MoveL 6678 to (240.69, 49.94, 97.46) mm, rotated rx -180 ry 0 rz 180 deg; joints [-31.755, 54.058, -83.161, 35.312, 114.429, 16.328]
  Call Extruder(210.56275)
  MoveL 6679 to (240.73, 50.24, 97.46) mm, rotated rx 180 ry 0 rz 180 deg; joints [-31.895, 54.08, -83.159, 35.455, 114.371, 16.375]
  MoveL 6680 to (240.73, 50.24, 97.46) mm, rotated rx 180 ry 0 rz 180 deg; joints [-31.895, 54.08, -83.159, 35.455, 114.371, 16.375]
  Call Extruder(210.72231)
  MoveL 6681 to (240.78, 50.55, 97.46) mm, rotated rx 180 ry 0 rz 180 deg; joints [-32.036, 54.101, -83.158, 35.597, 114.313, 16.422]
  MoveL 6682 to (240.78, 50.55, 97.46) mm, rotated rx 180 ry 0 rz 180 deg; joints [-32.036, 54.101, -83.158, 35.597, 114.313, 16.422]
  Call Extruder(210.88114)
  MoveL 6683 to (240.83, 50.86, 97.46) mm, rotated rx -180 ry 0 rz 180 deg; joints [-32.176, 54.122, -83.156, 35.738, 114.254, 16.468]
  MoveL 6684 to (240.83, 50.86, 97.46) mm, rotated rx -180 ry 0 rz 180 deg; joints [-32.176, 54.122, -83.156, 35.738, 114.254, 16.468]
  Call Extruder(211.05982)
  MoveL 6685 to (240.88, 51.2, 97.46) mm, rotated rx -180 ry 0 rz 180 deg; joints [-32.337, 54.146, -83.154, 35.9, 114.188, 16.521]
  MoveL 6686 to (240.88, 51.2, 97.46) mm, rotated rx -180 ry 0 rz 180 deg; joints [-32.337, 54.146, -83.154, 35.9, 114.188, 16.521]
  Call Extruder(211.25826)
  MoveL 6687 to (240.93, 51.59, 97.46) mm, rotated rx 180 ry 0 rz 180 deg; joints [-32.518, 54.171, -83.153, 36.083, 114.114, 16.58]
  MoveL 6688 to (240.93, 51.59, 97.46) mm, rotated rx 180 ry 0 rz 180 deg; joints [-32.518, 54.171, -83.153, 36.083, 114.114, 16.58]
  Call Extruder(211.45583)
  MoveL 6689 to (240.97, 51.98, 97.46) mm, rotated rx 180 ry 0 rz 180 deg; joints [-32.697, 54.197, -83.151, 36.264, 114.041, 16.639]
  MoveL 6690 to (240.97, 51.98, 97.46) mm, rotated rx 180 ry 0 rz 180 deg; joints [-32.697, 54.197, -83.151, 36.264, 114.041, 16.639]
  Call Extruder(211.65254)
  MoveL 6691 to (241.02, 52.36, 97.46) mm, rotated rx -180 ry 0 rz -180 deg; joints [-32.876, 54.223, -83.149, 36.445, 113.967, 16.698]
  MoveL 6692 to (241.02, 52.36, 97.46) mm, rotated rx -180 ry 0 rz -180 deg; joints [-32.876, 54.223, -83.149, 36.445, 113.967, 16.698]
  Call Extruder(211.84838)
  MoveL 6693 to (241.06, 52.75, 97.46) mm, rotated rx 180 ry 0 rz 180 deg; joints [-33.055, 54.249, -83.146, 36.624, 113.893, 16.755]
  MoveL 6694 to (241.06, 52.75, 97.46) mm, rotated rx 180 ry 0 rz 180 deg; joints [-33.055, 54.249, -83.146, 36.624, 113.893, 16.755]
  Call Extruder(212.14382)
  MoveL 6695 to (241.11, 53.34, 97.46) mm, rotated rx -180 ry 0 rz 180 deg; joints [-33.331, 54.287, -83.143, 36.903, 113.78, 16.845]
  MoveL 6696 to (241.11, 53.34, 97.46) mm, rotated rx -180 ry 0 rz 180 deg; joints [-33.331, 54.287, -83.143, 36.903, 113.78, 16.845]
  Call Extruder(212.43792)
  MoveL 6697 to (241.16, 53.93, 97.46) mm, rotated rx -180 ry 0 rz 180 deg; joints [-33.606, 54.325, -83.14, 37.179, 113.668, 16.934]
  MoveL 6698 to (241.16, 53.93, 97.46) mm, rotated rx -180 ry 0 rz 180 deg; joints [-33.606, 54.325, -83.14, 37.179, 113.668, 16.934]
  Call Extruder(212.73070)
  MoveL 6699 to (241.2, 54.52, 97.46) mm, rotated rx -180 ry 0 rz 180 deg; joints [-33.878, 54.363, -83.137, 37.452, 113.555, 17.021]
  MoveL 6700 to (241.2, 54.52, 97.46) mm, rotated rx -180 ry 0 rz 180 deg; joints [-33.878, 54.363, -83.137, 37.452, 113.555, 17.021]
  Call Extruder(213.30415)
  MoveL 6701 to (241.25, 55.68, 97.46) mm, rotated rx 180 ry 0 rz 180 deg; joints [-34.425, 54.435, -83.131, 38.001, 113.333, 17.195]
  MoveL 6702 to (241.25, 55.68, 97.46) mm, rotated rx 180 ry 0 rz 180 deg; joints [-34.425, 54.435, -83.131, 38.001, 113.333, 17.195]
  Call Extruder(214.01798)
  MoveL 6703 to (241.29, 57.14, 97.46) mm, rotated rx -180 ry 0 rz 180 deg; joints [-35.104, 54.524, -83.123, 38.681, 113.055, 17.407]
  Call Extruder(256.08287)
  MoveL 6704 to (241.29, 142.86, 97.46) mm, rotated rx 180 ry 0 rz 180 deg; joints [-60.361, 60.737, -81.719, 62.02, 100.2, 18.434]
  Call Extruder(256.51129)
  MoveL 6705 to (241.27, 143.73, 97.46) mm, rotated rx -180 ry 0 rz 180 deg; joints [-60.516, 60.803, -81.694, 62.155, 100.108, 18.379]
  MoveL 6706 to (241.27, 143.73, 97.46) mm, rotated rx -180 ry 0 rz 180 deg; joints [-60.516, 60.803, -81.694, 62.155, 100.108, 18.379]
  Call Extruder(257.08474)
  MoveL 6707 to (241.23, 144.9, 97.46) mm, rotated rx 180 ry 0 rz 180 deg; joints [-60.726, 60.888, -81.66, 62.34, 99.986, 18.307]
  MoveL 6708 to (241.23, 144.9, 97.46) mm, rotated rx 180 ry 0 rz 180 deg; joints [-60.726, 60.888, -81.66, 62.34, 99.986, 18.307]
  Call Extruder(257.51908)
  MoveL 6709 to (241.18, 145.77, 97.46) mm, rotated rx 180 ry 0 rz -180 deg; joints [-60.887, 60.952, -81.634, 62.481, 99.894, 18.253]
  MoveL 6710 to (241.18, 145.77, 97.46) mm, rotated rx 180 ry 0 rz -180 deg; joints [-60.887, 60.952, -81.634, 62.481, 99.894, 18.253]
  Call Extruder(257.81319)
  MoveL 6711 to (241.13, 146.36, 97.46) mm, rotated rx -180 ry 0 rz -180 deg; joints [-61, 60.995, -81.617, 62.58, 99.832, 18.218]
  MoveL 6712 to (241.13, 146.36, 97.46) mm, rotated rx -180 ry 0 rz -180 deg; joints [-61, 60.995, -81.617, 62.58, 99.832, 18.218]
  Call Extruder(258.10863)
  MoveL 6713 to (241.09, 146.95, 97.46) mm, rotated rx -180 ry 0 rz 180 deg; joints [-61.111, 61.037, -81.599, 62.678, 99.769, 18.182]
  MoveL 6714 to (241.09, 146.95, 97.46) mm, rotated rx -180 ry 0 rz 180 deg; joints [-61.111, 61.037, -81.599, 62.678, 99.769, 18.182]
  Call Extruder(258.35489)
  MoveL 6715 to (241.04, 147.44, 97.46) mm, rotated rx -180 ry 0 rz 180 deg; joints [-61.205, 61.072, -81.585, 62.761, 99.717, 18.153]
  MoveL 6716 to (241.04, 147.44, 97.46) mm, rotated rx -180 ry 0 rz 180 deg; joints [-61.205, 61.072, -81.585, 62.761, 99.717, 18.153]
  Call Extruder(258.55159)
  MoveL 6717 to (240.99, 147.83, 97.46) mm, rotated rx 180 ry 0 rz 180 deg; joints [-61.282, 61.099, -81.574, 62.83, 99.676, 18.131]
  MoveL 6718 to (240.99, 147.83, 97.46) mm, rotated rx 180 ry 0 rz 180 deg; joints [-61.282, 61.099, -81.574, 62.83, 99.676, 18.131]
  Call Extruder(258.74917)
  MoveL 6719 to (240.95, 148.22, 97.46) mm, rotated rx 180 ry 0 rz 180 deg; joints [-61.359, 61.127, -81.563, 62.898, 99.634, 18.109]
  MoveL 6720 to (240.95, 148.22, 97.46) mm, rotated rx 180 ry 0 rz 180 deg; joints [-61.359, 61.127, -81.563, 62.898, 99.634, 18.109]
  Call Extruder(258.94761)
  MoveL 6721 to (240.9, 148.6, 97.46) mm, rotated rx 180 ry 0 rz 180 deg; joints [-61.436, 61.154, -81.551, 62.966, 99.593, 18.086]
  MoveL 6722 to (240.9, 148.6, 97.46) mm, rotated rx 180 ry 0 rz 180 deg; joints [-61.436, 61.154, -81.551, 62.966, 99.593, 18.086]
  Call Extruder(259.14692)
  MoveL 6723 to (240.86, 148.99, 97.46) mm, rotated rx 180 ry 0 rz 180 deg; joints [-61.512, 61.181, -81.54, 63.033, 99.552, 18.064]
  MoveL 6724 to (240.86, 148.99, 97.46) mm, rotated rx 180 ry 0 rz 180 deg; joints [-61.512, 61.181, -81.54, 63.033, 99.552, 18.064]
  Call Extruder(259.30575)
  MoveL 6725 to (240.81, 149.3, 97.46) mm, rotated rx -180 ry 0 rz 180 deg; joints [-61.575, 61.202, -81.531, 63.09, 99.519, 18.047]
